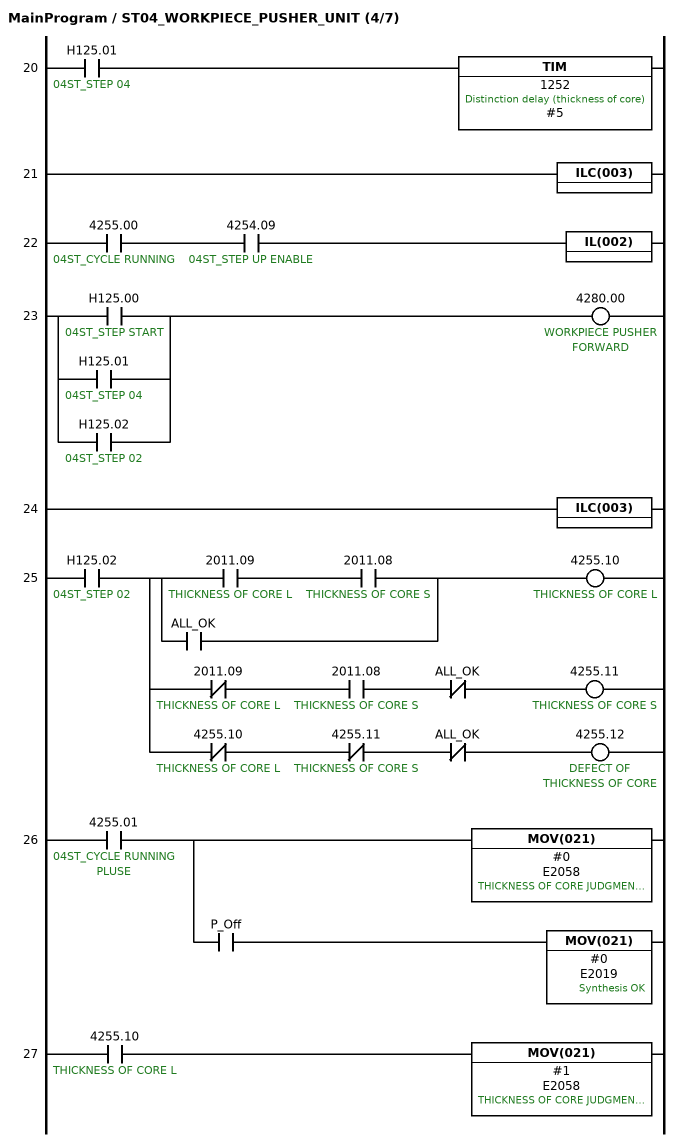
; [picture p336: MainProgram / ST04_WORKPIECE_PUSHER_UNIT, rungs 20-27]
; rung 20
LD H125.01  ; 04ST_STEP 04
TIM 1252 #5  ; Distinction delay (thickness of core)
; rung 21
ILC(003)
; rung 22
LD 4255.00  ; 04ST_CYCLE RUNNING
AND 4254.09  ; 04ST_STEP UP ENABLE
IL(002)
; rung 23
LD H125.00  ; 04ST_STEP START
OR H125.01  ; 04ST_STEP 04
OR H125.02  ; 04ST_STEP 02
OUT 4280.00  ; WORKPIECE PUSHER FORWARD
; rung 24
ILC(003)
; rung 25
LD H125.02  ; 04ST_STEP 02
OUT TR0
LD 2011.09  ; THICKNESS OF CORE L
AND 2011.08  ; THICKNESS OF CORE S
OR ALL_OK
ANDLD
OUT 4255.10  ; THICKNESS OF CORE L
LD TR0
ANDNOT 2011.09  ; THICKNESS OF CORE L
AND 2011.08  ; THICKNESS OF CORE S
ANDNOT ALL_OK
OUT 4255.11  ; THICKNESS OF CORE S
LD TR0
ANDNOT 4255.10  ; THICKNESS OF CORE L
ANDNOT 4255.11  ; THICKNESS OF CORE S
ANDNOT ALL_OK
OUT 4255.12  ; DEFECT OF THICKNESS OF CORE
; rung 26
LD 4255.01  ; 04ST_CYCLE RUNNING PLUSE
MOV(021) #0 E2058  ; THICKNESS OF CORE JUDGMENT RESULT (1:L , 2: S)
AND P_Off
MOV(021) #0 E2019  ; Synthesis OK
; rung 27
LD 4255.10  ; THICKNESS OF CORE L
MOV(021) #1 E2058  ; THICKNESS OF CORE JUDGMENT RESULT (1:L , 2: S)

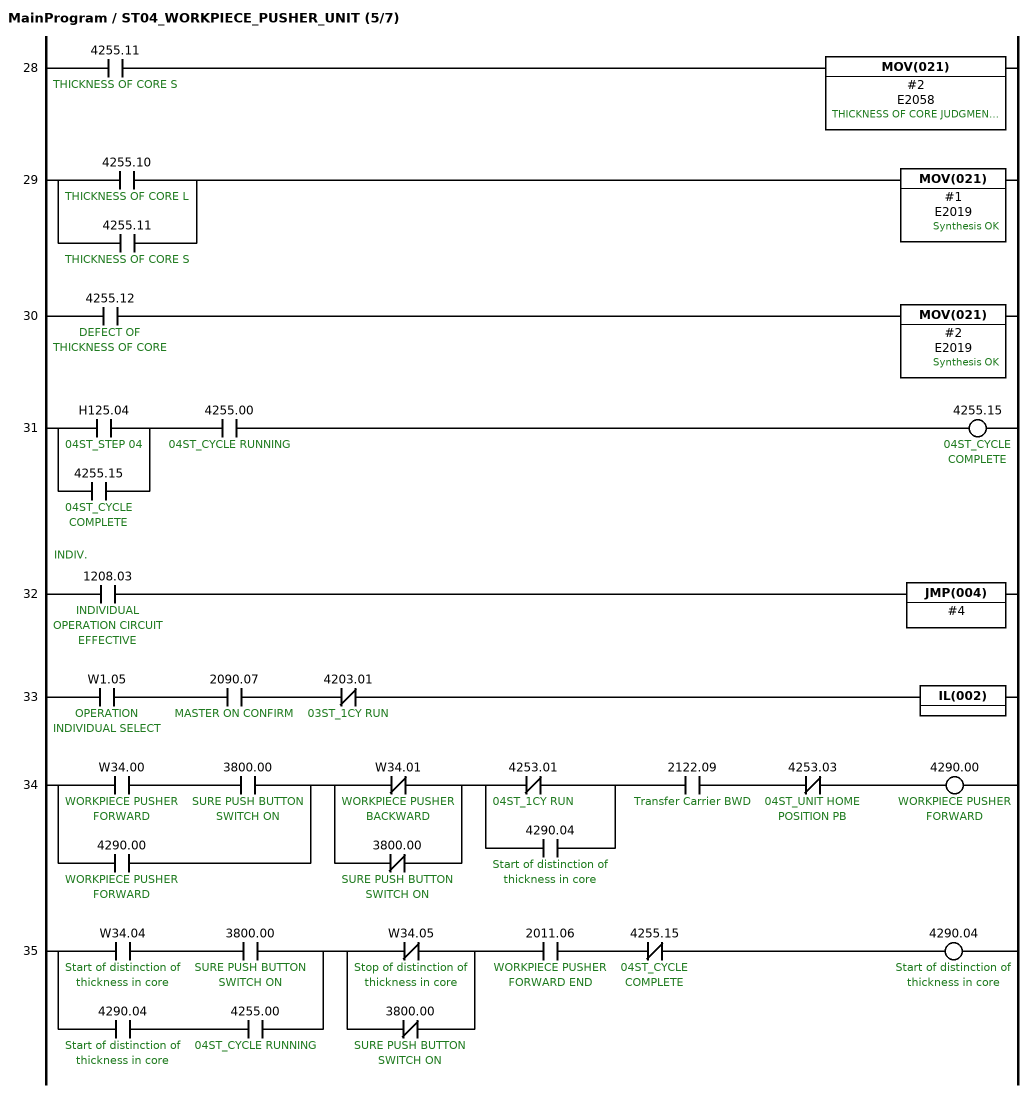
; rung 28
LD 4255.11  ; THICKNESS OF CORE S
MOV(021) #2 E2058  ; THICKNESS OF CORE JUDGMENT RESULT (1:L , 2: S)
; rung 29
LD 4255.10  ; THICKNESS OF CORE L
OR 4255.11  ; THICKNESS OF CORE S
MOV(021) #1 E2019  ; Synthesis OK
; rung 30
LD 4255.12  ; DEFECT OF THICKNESS OF CORE
MOV(021) #2 E2019  ; Synthesis OK
; rung 31
LD H125.04  ; 04ST_STEP 04
OR 4255.15  ; 04ST_CYCLE COMPLETE
AND 4255.00  ; 04ST_CYCLE RUNNING
OUT 4255.15  ; 04ST_CYCLE COMPLETE
; rung 32: INDIV.
LD 1208.03  ; INDIVIDUAL OPERATION CIRCUIT EFFECTIVE
JMP(004) #4
; rung 33
LD W1.05  ; OPERATION INDIVIDUAL SELECT
AND 2090.07  ; MASTER ON CONFIRM
ANDNOT 4203.01  ; 03ST_1CY RUN
IL(002)
; rung 34
LD W34.00  ; WORKPIECE PUSHER FORWARD
AND 3800.00  ; SURE PUSH BUTTON SWITCH ON
OR 4290.00  ; WORKPIECE PUSHER FORWARD
LDNOT W34.01  ; WORKPIECE PUSHER BACKWARD
ORNOT 3800.00  ; SURE PUSH BUTTON SWITCH ON
ANDLD
LDNOT 4253.01  ; 04ST_1CY RUN
OR 4290.04  ; Start of distinction of thickness in core
ANDLD
AND 2122.09  ; Transfer Carrier BWD
ANDNOT 4253.03  ; 04ST_UNIT HOME POSITION PB
OUT 4290.00  ; WORKPIECE PUSHER FORWARD
; rung 35
LD W34.04  ; Start of distinction of thickness in core
AND 3800.00  ; SURE PUSH BUTTON SWITCH ON
LD 4290.04  ; Start of distinction of thickness in core
AND 4255.00  ; 04ST_CYCLE RUNNING
ORLD
LDNOT W34.05  ; Stop of distinction of thickness in core
ORNOT 3800.00  ; SURE PUSH BUTTON SWITCH ON
ANDLD
AND 2011.06  ; WORKPIECE PUSHER FORWARD END
ANDNOT 4255.15  ; 04ST_CYCLE COMPLETE
OUT 4290.04  ; Start of distinction of thickness in core

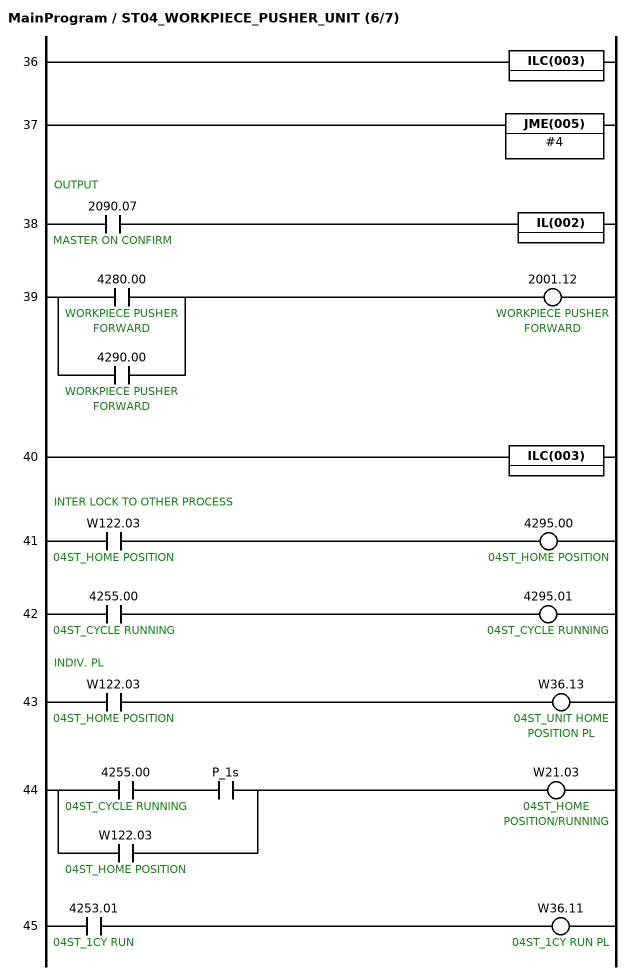
; rung 36
ILC(003)
; rung 37
JME(005) #4
; rung 38: OUTPUT
LD 2090.07  ; MASTER ON CONFIRM
IL(002)
; rung 39
LD 4280.00  ; WORKPIECE PUSHER FORWARD
OR 4290.00  ; WORKPIECE PUSHER FORWARD
OUT 2001.12  ; WORKPIECE PUSHER FORWARD
; rung 40
ILC(003)
; rung 41: INTER LOCK TO OTHER PROCESS
LD W122.03  ; 04ST_HOME POSITION
OUT 4295.00  ; 04ST_HOME POSITION
; rung 42
LD 4255.00  ; 04ST_CYCLE RUNNING
OUT 4295.01  ; 04ST_CYCLE RUNNING
; rung 43: INDIV. PL
LD W122.03  ; 04ST_HOME POSITION
OUT W36.13  ; 04ST_UNIT HOME POSITION PL
; rung 44
LD 4255.00  ; 04ST_CYCLE RUNNING
AND P_1s
OR W122.03  ; 04ST_HOME POSITION
OUT W21.03  ; 04ST_HOME POSITION/RUNNING
; rung 45
LD 4253.01  ; 04ST_1CY RUN
OUT W36.11  ; 04ST_1CY RUN PL

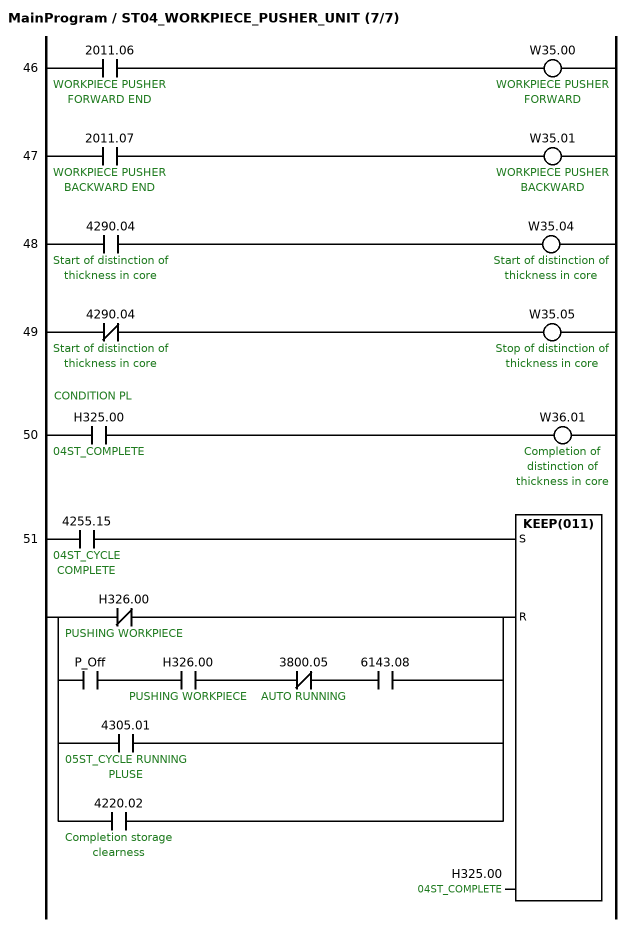
; rung 46
LD 2011.06  ; WORKPIECE PUSHER FORWARD END
OUT W35.00  ; WORKPIECE PUSHER FORWARD
; rung 47
LD 2011.07  ; WORKPIECE PUSHER BACKWARD END
OUT W35.01  ; WORKPIECE PUSHER BACKWARD
; rung 48
LD 4290.04  ; Start of distinction of thickness in core
OUT W35.04  ; Start of distinction of thickness in core
; rung 49
LDNOT 4290.04  ; Start of distinction of thickness in core
OUT W35.05  ; Stop of distinction of thickness in core
; rung 50: CONDITION PL
LD H325.00  ; 04ST_COMPLETE
OUT W36.01  ; Completion of distinction of thickness in core
; rung 51
LD 4255.15  ; 04ST_CYCLE COMPLETE
LDNOT H326.00  ; PUSHING WORKPIECE
LD P_Off
AND H326.00  ; PUSHING WORKPIECE
ANDNOT 3800.05  ; AUTO RUNNING
AND 6143.08
ORLD
OR 4305.01  ; 05ST_CYCLE RUNNING PLUSE
OR 4220.02  ; Completion storage clearness
KEEP(011) H325.00  ; 04ST_COMPLETE

### Section ST05_INSULATION_TEST_UNIT

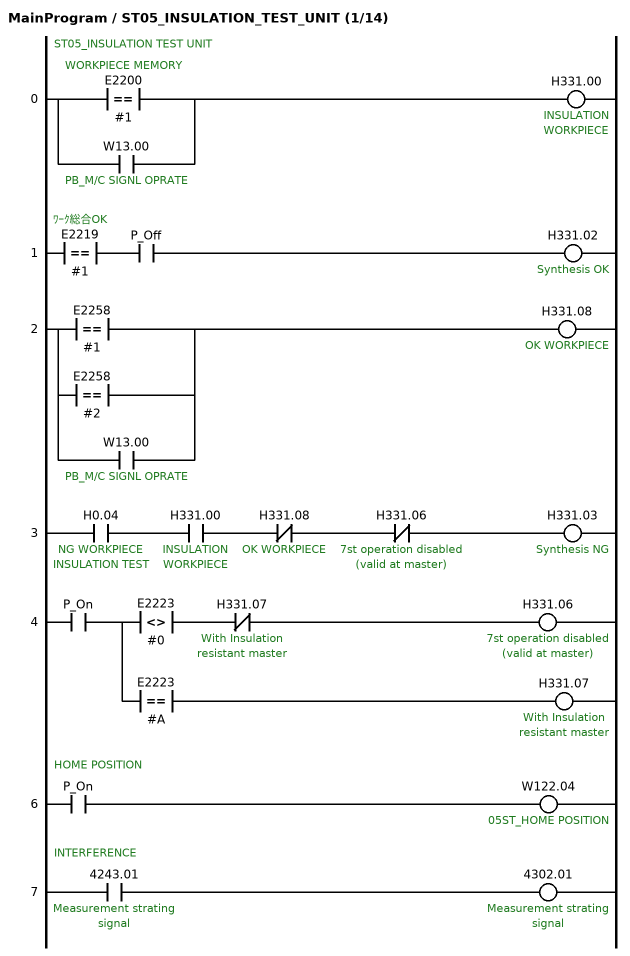
; rung 0: ST05_INSULATION TEST UNIT
LD=(300) E2200 #1  ; WORKPIECE MEMORY
OR W13.00  ; PB_M/C SIGNL OPRATE
OUT H331.00  ; INSULATION WORKPIECE
; rung 1
LD=(300) E2219 #1  ; ﾜｰｸ総合OK
AND P_Off
OUT H331.02  ; Synthesis OK
; rung 2
LD=(300) E2258 #1
OR=(300) E2258 #2
OR W13.00  ; PB_M/C SIGNL OPRATE
OUT H331.08  ; OK WORKPIECE
; rung 3
LD H0.04  ; NG WORKPIECE INSULATION TEST
AND H331.00  ; INSULATION WORKPIECE
ANDNOT H331.08  ; OK WORKPIECE
ANDNOT H331.06  ; 7st operation disabled (valid at master)
OUT H331.03  ; Synthesis NG
; rung 4
LD P_On
OUT TR0
AND<>(305) E2223 #0
ANDNOT H331.07  ; With Insulation resistant master
OUT H331.06  ; 7st operation disabled (valid at master)
LD TR0
AND=(300) E2223 #A
OUT H331.07  ; With Insulation resistant master
; rung 5: TIMER
; rung 6: HOME POSITION
LD P_On
OUT W122.04  ; 05ST_HOME POSITION
; rung 7: INTERFERENCE
LD 4243.01  ; Measurement strating signal
OUT 4302.01  ; Measurement strating signal

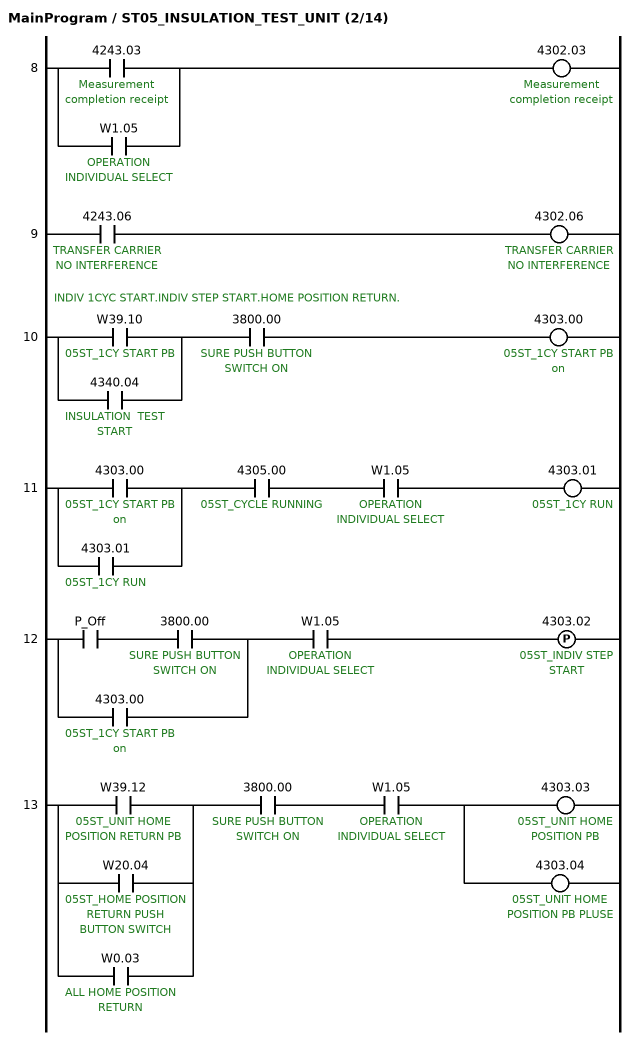
; rung 8
LD 4243.03  ; Measurement completion receipt
OR W1.05  ; OPERATION INDIVIDUAL SELECT
OUT 4302.03  ; Measurement completion receipt
; rung 9
LD 4243.06  ; TRANSFER CARRIER NO INTERFERENCE
OUT 4302.06  ; TRANSFER CARRIER NO INTERFERENCE
; rung 10: INDIV 1CYC START.INDIV STEP START.HOME POSITION RETURN.
LD W39.10  ; 05ST_1CY START PB
OR 4340.04  ; INSULATION  TEST START
AND 3800.00  ; SURE PUSH BUTTON SWITCH ON
OUT 4303.00  ; 05ST_1CY START PB on
; rung 11
LD 4303.00  ; 05ST_1CY START PB on
OR 4303.01  ; 05ST_1CY RUN
AND 4305.00  ; 05ST_CYCLE RUNNING
AND W1.05  ; OPERATION INDIVIDUAL SELECT
OUT 4303.01  ; 05ST_1CY RUN
; rung 12
LD P_Off
AND 3800.00  ; SURE PUSH BUTTON SWITCH ON
OR 4303.00  ; 05ST_1CY START PB on
AND W1.05  ; OPERATION INDIVIDUAL SELECT
DIFU(013) 4303.02  ; 05ST_INDIV STEP START
; rung 13
LD W39.12  ; 05ST_UNIT HOME POSITION RETURN PB
OR W20.04  ; 05ST_HOME POSITION RETURN PUSH BUTTON SWITCH
OR W0.03  ; ALL HOME POSITION RETURN
AND 3800.00  ; SURE PUSH BUTTON SWITCH ON
AND W1.05  ; OPERATION INDIVIDUAL SELECT
OUT 4303.03  ; 05ST_UNIT HOME POSITION PB
OUT 4303.04  ; 05ST_UNIT HOME POSITION PB PLUSE

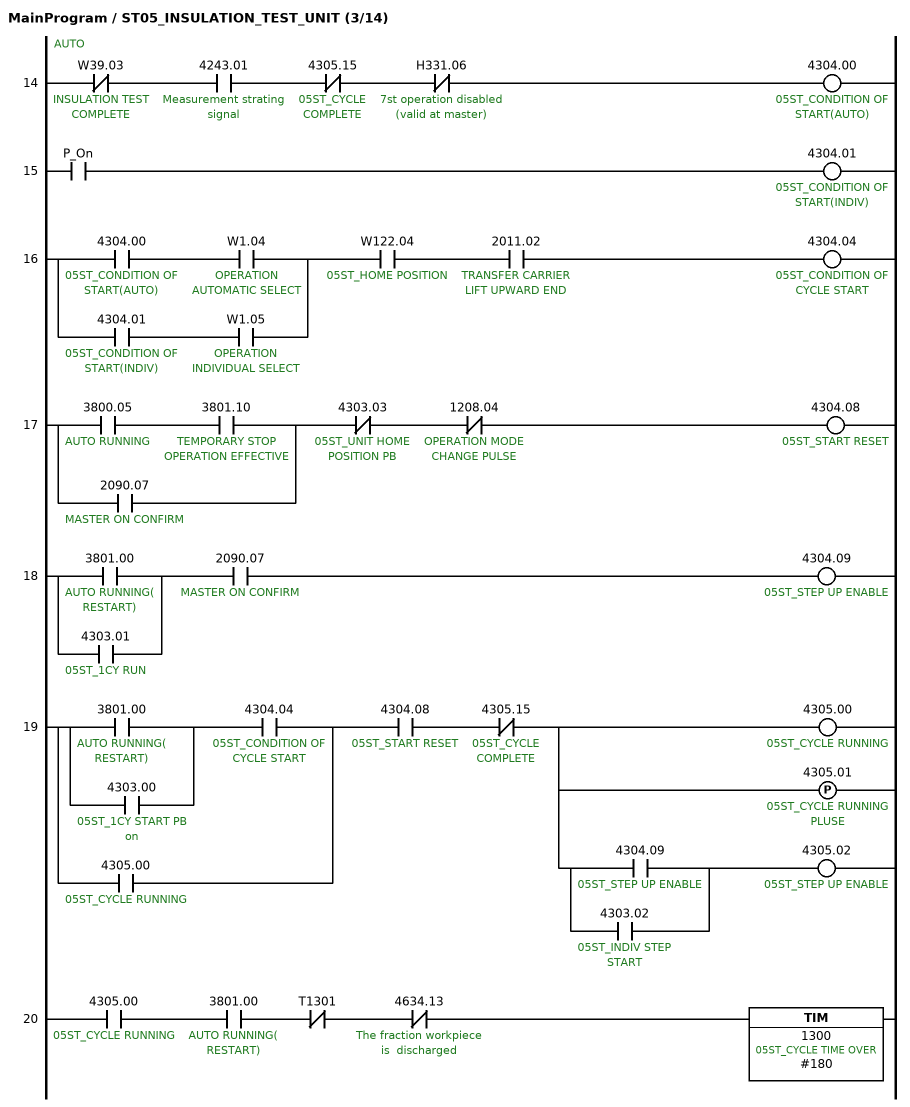
; rung 14: AUTO
LDNOT W39.03  ; INSULATION TEST COMPLETE
AND 4243.01  ; Measurement strating signal
ANDNOT 4305.15  ; 05ST_CYCLE COMPLETE
ANDNOT H331.06  ; 7st operation disabled (valid at master)
OUT 4304.00  ; 05ST_CONDITION OF START(AUTO)
; rung 15
LD P_On
OUT 4304.01  ; 05ST_CONDITION OF START(INDIV)
; rung 16
LD 4304.00  ; 05ST_CONDITION OF START(AUTO)
AND W1.04  ; OPERATION AUTOMATIC SELECT
LD 4304.01  ; 05ST_CONDITION OF START(INDIV)
AND W1.05  ; OPERATION INDIVIDUAL SELECT
ORLD
AND W122.04  ; 05ST_HOME POSITION
AND 2011.02  ; TRANSFER CARRIER LIFT UPWARD END
OUT 4304.04  ; 05ST_CONDITION OF CYCLE START
; rung 17
LD 3800.05  ; AUTO RUNNING
AND 3801.10  ; TEMPORARY STOP OPERATION EFFECTIVE
OR 2090.07  ; MASTER ON CONFIRM
ANDNOT 4303.03  ; 05ST_UNIT HOME POSITION PB
ANDNOT 1208.04  ; OPERATION MODE CHANGE PULSE
OUT 4304.08  ; 05ST_START RESET
; rung 18
LD 3801.00  ; AUTO RUNNING(RESTART)
OR 4303.01  ; 05ST_1CY RUN
AND 2090.07  ; MASTER ON CONFIRM
OUT 4304.09  ; 05ST_STEP UP ENABLE
; rung 19
LD 3801.00  ; AUTO RUNNING(RESTART)
OR 4303.00  ; 05ST_1CY START PB on
AND 4304.04  ; 05ST_CONDITION OF CYCLE START
OR 4305.00  ; 05ST_CYCLE RUNNING
AND 4304.08  ; 05ST_START RESET
ANDNOT 4305.15  ; 05ST_CYCLE COMPLETE
OUT 4305.00  ; 05ST_CYCLE RUNNING
DIFU(013) 4305.01  ; 05ST_CYCLE RUNNING PLUSE
LD 4304.09  ; 05ST_STEP UP ENABLE
OR 4303.02  ; 05ST_INDIV STEP START
ANDLD
OUT 4305.02  ; 05ST_STEP UP ENABLE
; rung 20
LD 4305.00  ; 05ST_CYCLE RUNNING
AND 3801.00  ; AUTO RUNNING(RESTART)
ANDNOT T1301
ANDNOT 4634.13  ; The fraction workpiece is  discharged
TIM 1300 #180  ; 05ST_CYCLE TIME OVER

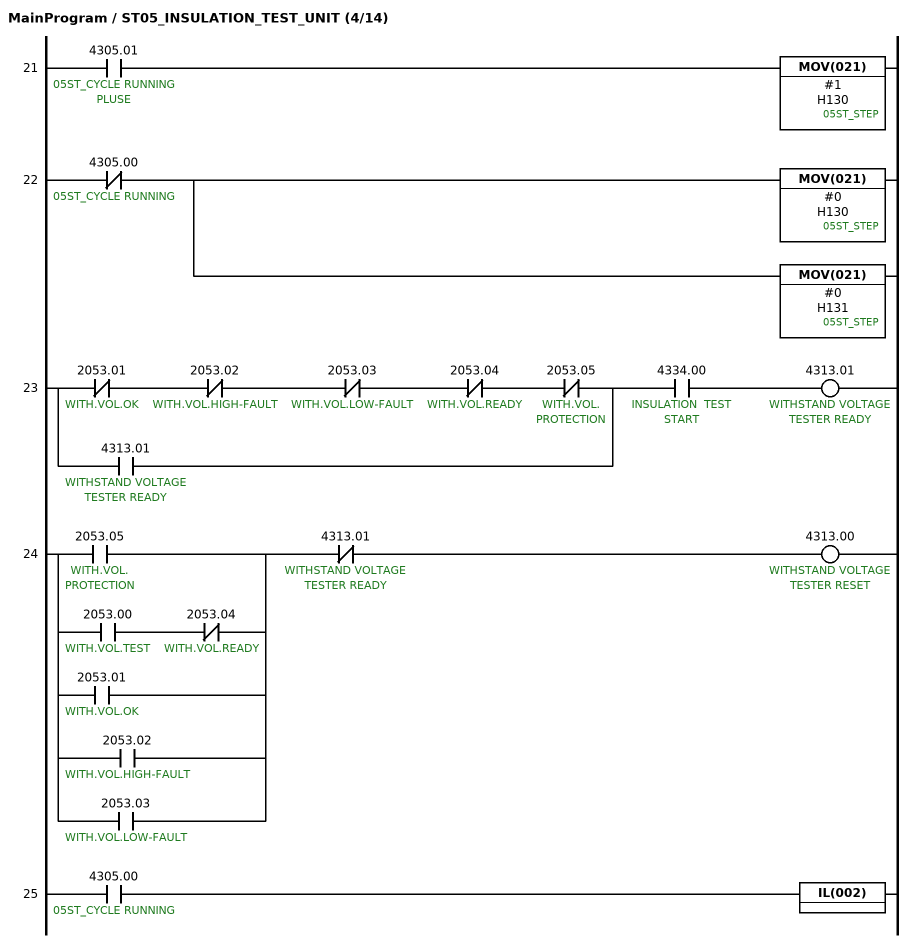
; rung 21
LD 4305.01  ; 05ST_CYCLE RUNNING PLUSE
MOV(021) #1 H130  ; 05ST_STEP
; rung 22
LDNOT 4305.00  ; 05ST_CYCLE RUNNING
MOV(021) #0 H130  ; 05ST_STEP
MOV(021) #0 H131  ; 05ST_STEP
; rung 23
LDNOT 2053.01  ; WITH.VOL.OK
ANDNOT 2053.02  ; WITH.VOL.HIGH-FAULT
ANDNOT 2053.03  ; WITH.VOL.LOW-FAULT
ANDNOT 2053.04  ; WITH.VOL.READY
ANDNOT 2053.05  ; WITH.VOL.PROTECTION
OR 4313.01  ; WITHSTAND VOLTAGE TESTER READY
AND 4334.00  ; INSULATION  TEST START
OUT 4313.01  ; WITHSTAND VOLTAGE TESTER READY
; rung 24
LD 2053.05  ; WITH.VOL.PROTECTION
LD 2053.00  ; WITH.VOL.TEST
ANDNOT 2053.04  ; WITH.VOL.READY
ORLD
OR 2053.01  ; WITH.VOL.OK
OR 2053.02  ; WITH.VOL.HIGH-FAULT
OR 2053.03  ; WITH.VOL.LOW-FAULT
ANDNOT 4313.01  ; WITHSTAND VOLTAGE TESTER READY
OUT 4313.00  ; WITHSTAND VOLTAGE TESTER RESET
; rung 25
LD 4305.00  ; 05ST_CYCLE RUNNING
IL(002)

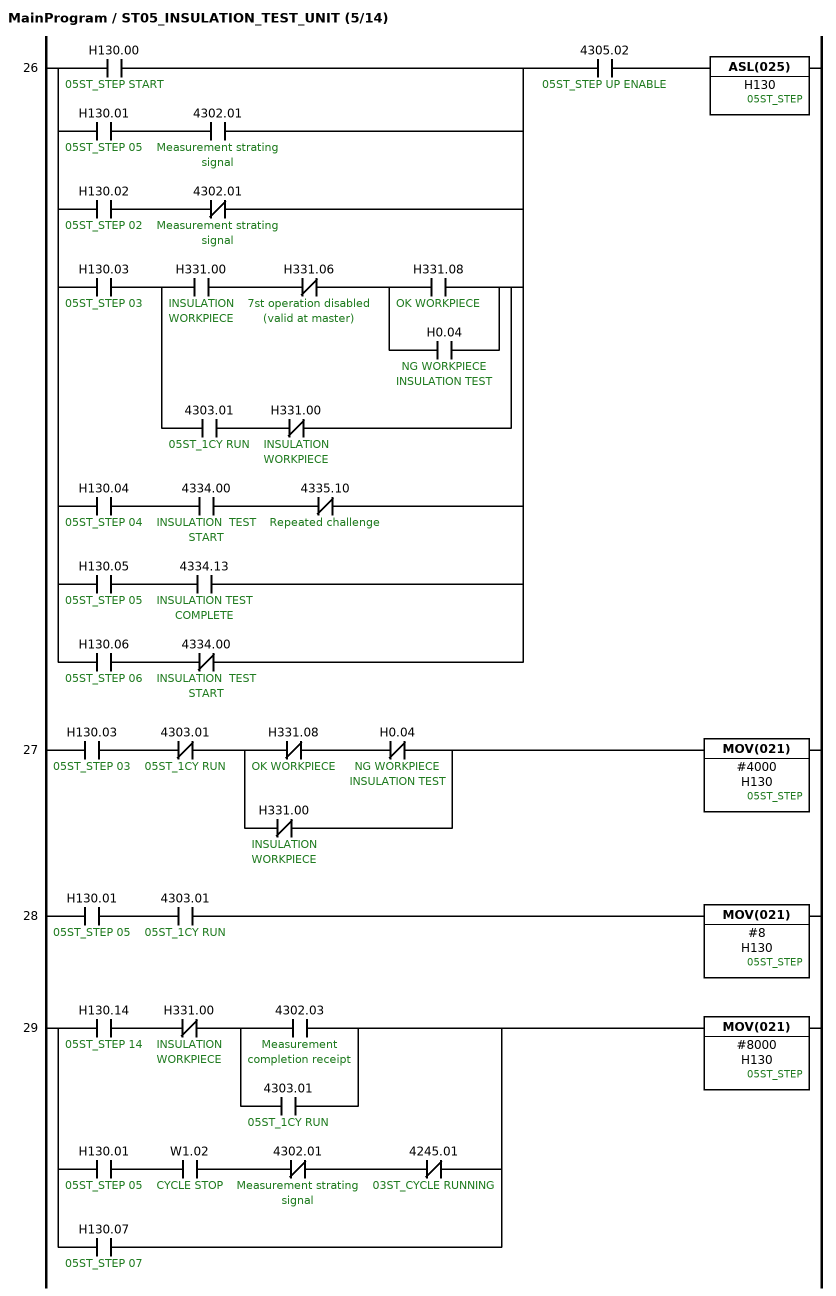
; rung 26
LD H130.00  ; 05ST_STEP START
LD H130.01  ; 05ST_STEP 05
AND 4302.01  ; Measurement strating signal
ORLD
LD H130.02  ; 05ST_STEP 02
ANDNOT 4302.01  ; Measurement strating signal
ORLD
LD H130.03  ; 05ST_STEP 03
LD H331.00  ; INSULATION WORKPIECE
ANDNOT H331.06  ; 7st operation disabled (valid at master)
LD H331.08  ; OK WORKPIECE
OR H0.04  ; NG WORKPIECE INSULATION TEST
ANDLD
LD 4303.01  ; 05ST_1CY RUN
ANDNOT H331.00  ; INSULATION WORKPIECE
ORLD
ANDLD
ORLD
LD H130.04  ; 05ST_STEP 04
AND 4334.00  ; INSULATION  TEST START
ANDNOT 4335.10  ; Repeated challenge
ORLD
LD H130.05  ; 05ST_STEP 05
AND 4334.13  ; INSULATION TEST COMPLETE
ORLD
LD H130.06  ; 05ST_STEP 06
ANDNOT 4334.00  ; INSULATION  TEST START
ORLD
AND 4305.02  ; 05ST_STEP UP ENABLE
ASL(025) H130  ; 05ST_STEP
; rung 27
LD H130.03  ; 05ST_STEP 03
ANDNOT 4303.01  ; 05ST_1CY RUN
LDNOT H331.08  ; OK WORKPIECE
ANDNOT H0.04  ; NG WORKPIECE INSULATION TEST
ORNOT H331.00  ; INSULATION WORKPIECE
ANDLD
MOV(021) #4000 H130  ; 05ST_STEP
; rung 28
LD H130.01  ; 05ST_STEP 05
AND 4303.01  ; 05ST_1CY RUN
MOV(021) #8 H130  ; 05ST_STEP
; rung 29
LD H130.14  ; 05ST_STEP 14
ANDNOT H331.00  ; INSULATION WORKPIECE
LD 4302.03  ; Measurement completion receipt
OR 4303.01  ; 05ST_1CY RUN
ANDLD
LD H130.01  ; 05ST_STEP 05
AND W1.02  ; CYCLE STOP
ANDNOT 4302.01  ; Measurement strating signal
ANDNOT 4245.01  ; 03ST_CYCLE RUNNING
ORLD
OR H130.07  ; 05ST_STEP 07
MOV(021) #8000 H130  ; 05ST_STEP

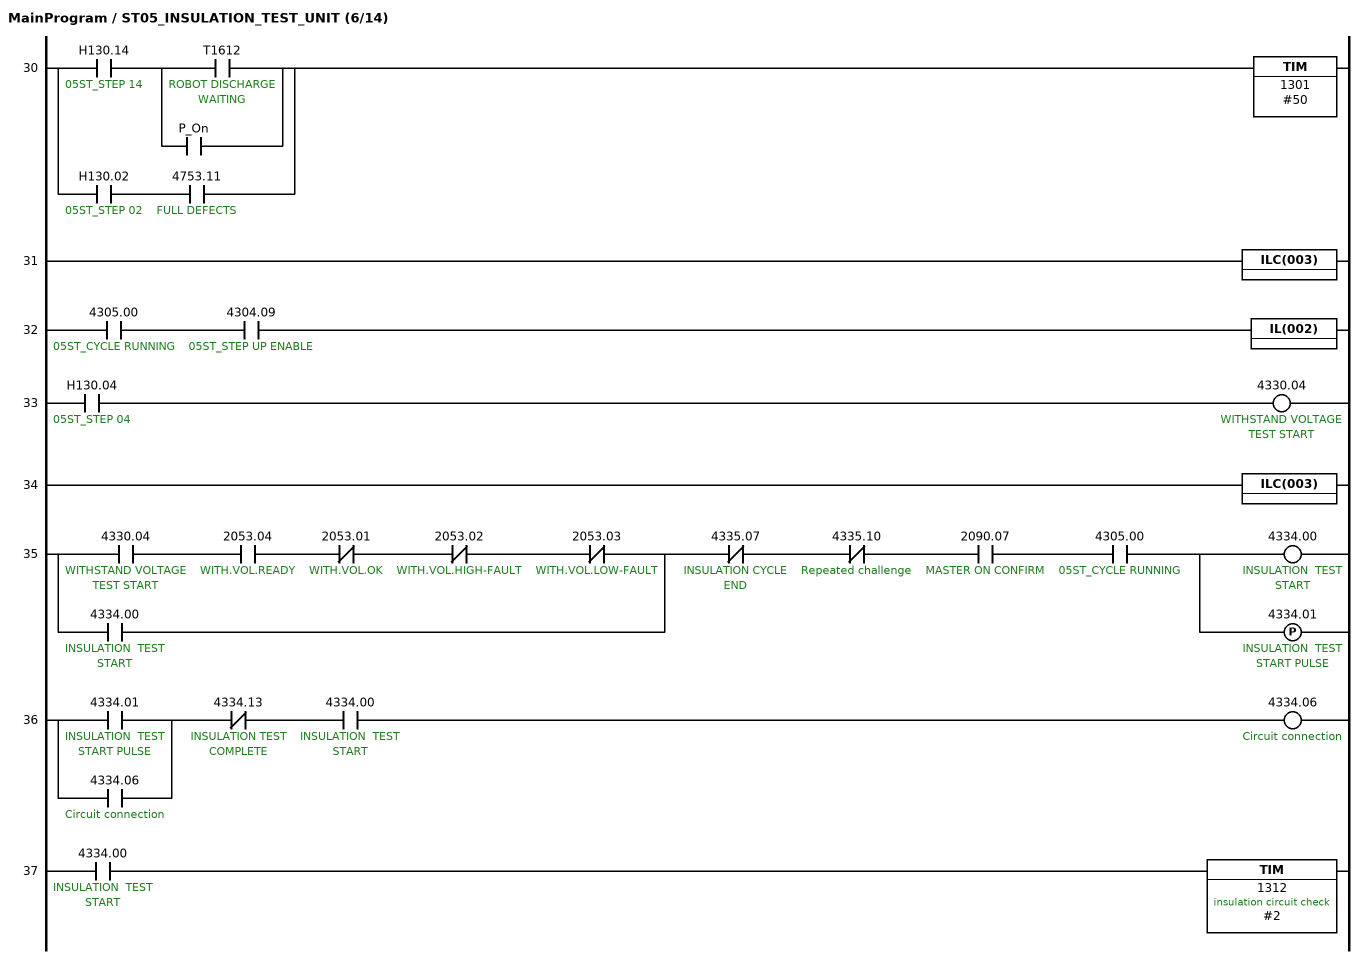
; rung 30
LD H130.14  ; 05ST_STEP 14
LD T1612  ; ROBOT DISCHARGE WAITING
OR P_On
ANDLD
LD H130.02  ; 05ST_STEP 02
AND 4753.11  ; FULL DEFECTS
ORLD
TIM 1301 #50
; rung 31
ILC(003)
; rung 32
LD 4305.00  ; 05ST_CYCLE RUNNING
AND 4304.09  ; 05ST_STEP UP ENABLE
IL(002)
; rung 33
LD H130.04  ; 05ST_STEP 04
OUT 4330.04  ; WITHSTAND VOLTAGE TEST START
; rung 34
ILC(003)
; rung 35
LD 4330.04  ; WITHSTAND VOLTAGE TEST START
AND 2053.04  ; WITH.VOL.READY
ANDNOT 2053.01  ; WITH.VOL.OK
ANDNOT 2053.02  ; WITH.VOL.HIGH-FAULT
ANDNOT 2053.03  ; WITH.VOL.LOW-FAULT
OR 4334.00  ; INSULATION  TEST START
ANDNOT 4335.07  ; INSULATION CYCLE END
ANDNOT 4335.10  ; Repeated challenge
AND 2090.07  ; MASTER ON CONFIRM
AND 4305.00  ; 05ST_CYCLE RUNNING
OUT 4334.00  ; INSULATION  TEST START
DIFU(013) 4334.01  ; INSULATION  TEST START PULSE
; rung 36
LD 4334.01  ; INSULATION  TEST START PULSE
OR 4334.06  ; Circuit connection
ANDNOT 4334.13  ; INSULATION TEST COMPLETE
AND 4334.00  ; INSULATION  TEST START
OUT 4334.06  ; Circuit connection
; rung 37
LD 4334.00  ; INSULATION  TEST START
TIM 1312 #2  ; insulation circuit check

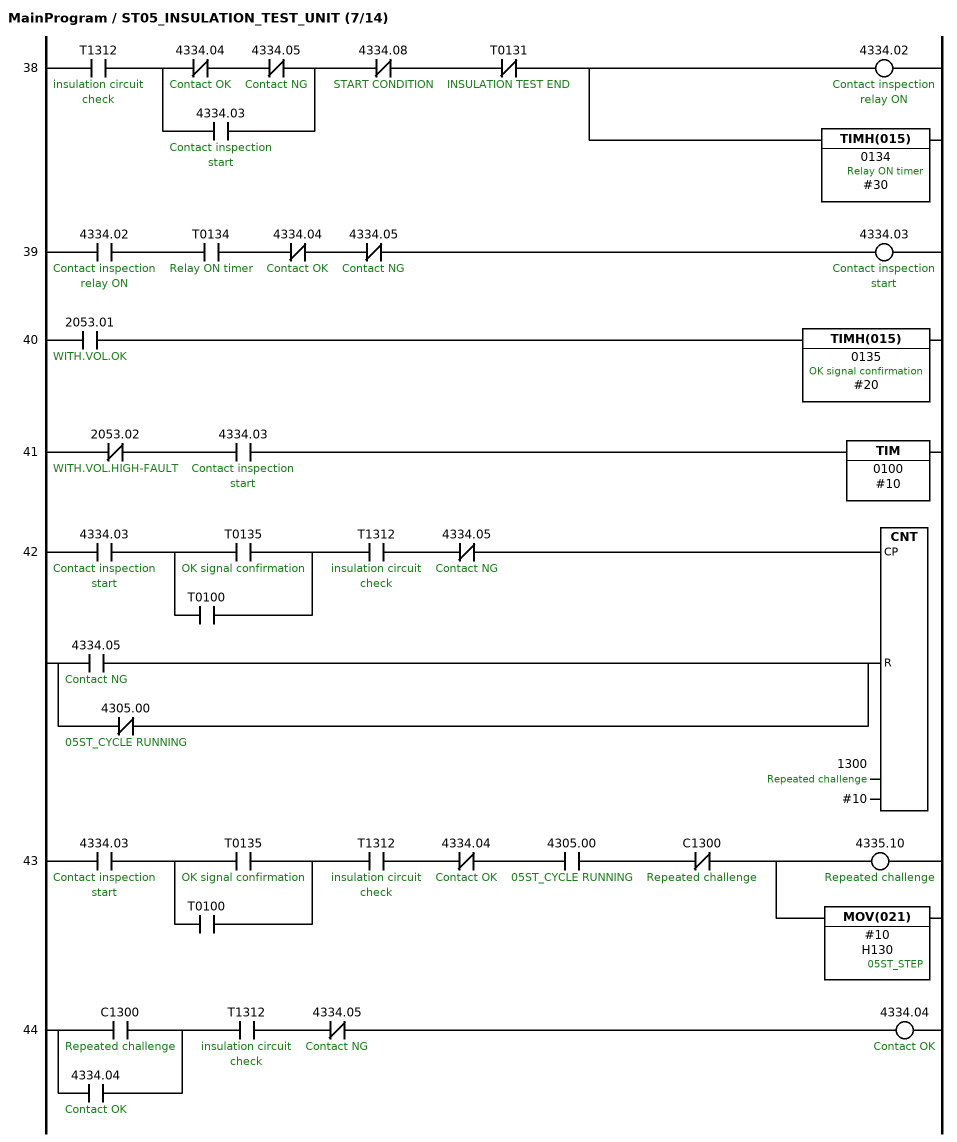
; rung 38
LD T1312  ; insulation circuit check
LDNOT 4334.04  ; Contact OK
ANDNOT 4334.05  ; Contact NG
OR 4334.03  ; Contact inspection start
ANDLD
ANDNOT 4334.08  ; START CONDITION
ANDNOT T0131  ; INSULATION TEST END
OUT 4334.02  ; Contact inspection relay ON
TIMH(015) 0134 #30  ; Relay ON timer
; rung 39
LD 4334.02  ; Contact inspection relay ON
AND T0134  ; Relay ON timer
ANDNOT 4334.04  ; Contact OK
ANDNOT 4334.05  ; Contact NG
OUT 4334.03  ; Contact inspection start
; rung 40
LD 2053.01  ; WITH.VOL.OK
TIMH(015) 0135 #20  ; OK signal confirmation
; rung 41
LDNOT 2053.02  ; WITH.VOL.HIGH-FAULT
AND 4334.03  ; Contact inspection start
TIM 0100 #10
; rung 42
LD 4334.03  ; Contact inspection start
LD T0135  ; OK signal confirmation
OR T0100
ANDLD
AND T1312  ; insulation circuit check
ANDNOT 4334.05  ; Contact NG
LD 4334.05  ; Contact NG
ORNOT 4305.00  ; 05ST_CYCLE RUNNING
CNT 1300 #10  ; Repeated challenge
; rung 43
LD 4334.03  ; Contact inspection start
LD T0135  ; OK signal confirmation
OR T0100
ANDLD
AND T1312  ; insulation circuit check
ANDNOT 4334.04  ; Contact OK
AND 4305.00  ; 05ST_CYCLE RUNNING
ANDNOT C1300  ; Repeated challenge
OUT 4335.10  ; Repeated challenge
MOV(021) #10 H130  ; 05ST_STEP
; rung 44
LD C1300  ; Repeated challenge
OR 4334.04  ; Contact OK
AND T1312  ; insulation circuit check
ANDNOT 4334.05  ; Contact NG
OUT 4334.04  ; Contact OK

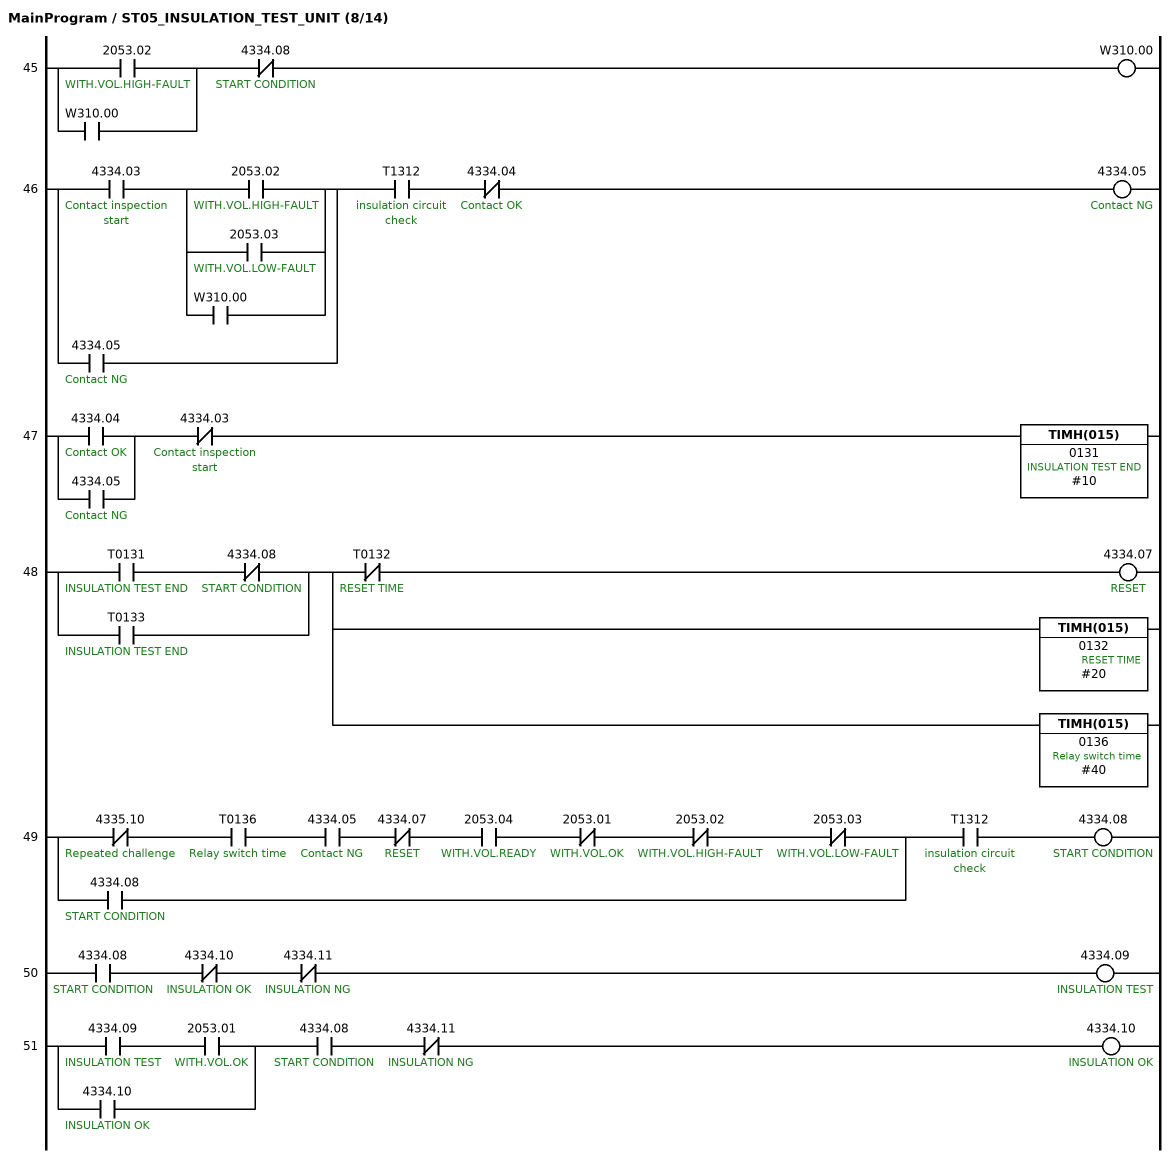
; rung 45
LD 2053.02  ; WITH.VOL.HIGH-FAULT
OR W310.00
ANDNOT 4334.08  ; START CONDITION
OUT W310.00
; rung 46
LD 4334.03  ; Contact inspection start
LD 2053.02  ; WITH.VOL.HIGH-FAULT
OR 2053.03  ; WITH.VOL.LOW-FAULT
OR W310.00
ANDLD
OR 4334.05  ; Contact NG
AND T1312  ; insulation circuit check
ANDNOT 4334.04  ; Contact OK
OUT 4334.05  ; Contact NG
; rung 47
LD 4334.04  ; Contact OK
OR 4334.05  ; Contact NG
ANDNOT 4334.03  ; Contact inspection start
TIMH(015) 0131 #10  ; INSULATION TEST END
; rung 48
LD T0131  ; INSULATION TEST END
ANDNOT 4334.08  ; START CONDITION
OR T0133  ; INSULATION TEST END
OUT TR0
ANDNOT T0132  ; RESET TIME
OUT 4334.07  ; RESET
LD TR0
TIMH(015) 0132 #20  ; RESET TIME
TIMH(015) 0136 #40  ; Relay switch time
; rung 49
LDNOT 4335.10  ; Repeated challenge
AND T0136  ; Relay switch time
AND 4334.05  ; Contact NG
ANDNOT 4334.07  ; RESET
AND 2053.04  ; WITH.VOL.READY
ANDNOT 2053.01  ; WITH.VOL.OK
ANDNOT 2053.02  ; WITH.VOL.HIGH-FAULT
ANDNOT 2053.03  ; WITH.VOL.LOW-FAULT
OR 4334.08  ; START CONDITION
AND T1312  ; insulation circuit check
OUT 4334.08  ; START CONDITION
; rung 50
LD 4334.08  ; START CONDITION
ANDNOT 4334.10  ; INSULATION OK
ANDNOT 4334.11  ; INSULATION NG
OUT 4334.09  ; INSULATION TEST
; rung 51
LD 4334.09  ; INSULATION TEST
AND 2053.01  ; WITH.VOL.OK
OR 4334.10  ; INSULATION OK
AND 4334.08  ; START CONDITION
ANDNOT 4334.11  ; INSULATION NG
OUT 4334.10  ; INSULATION OK

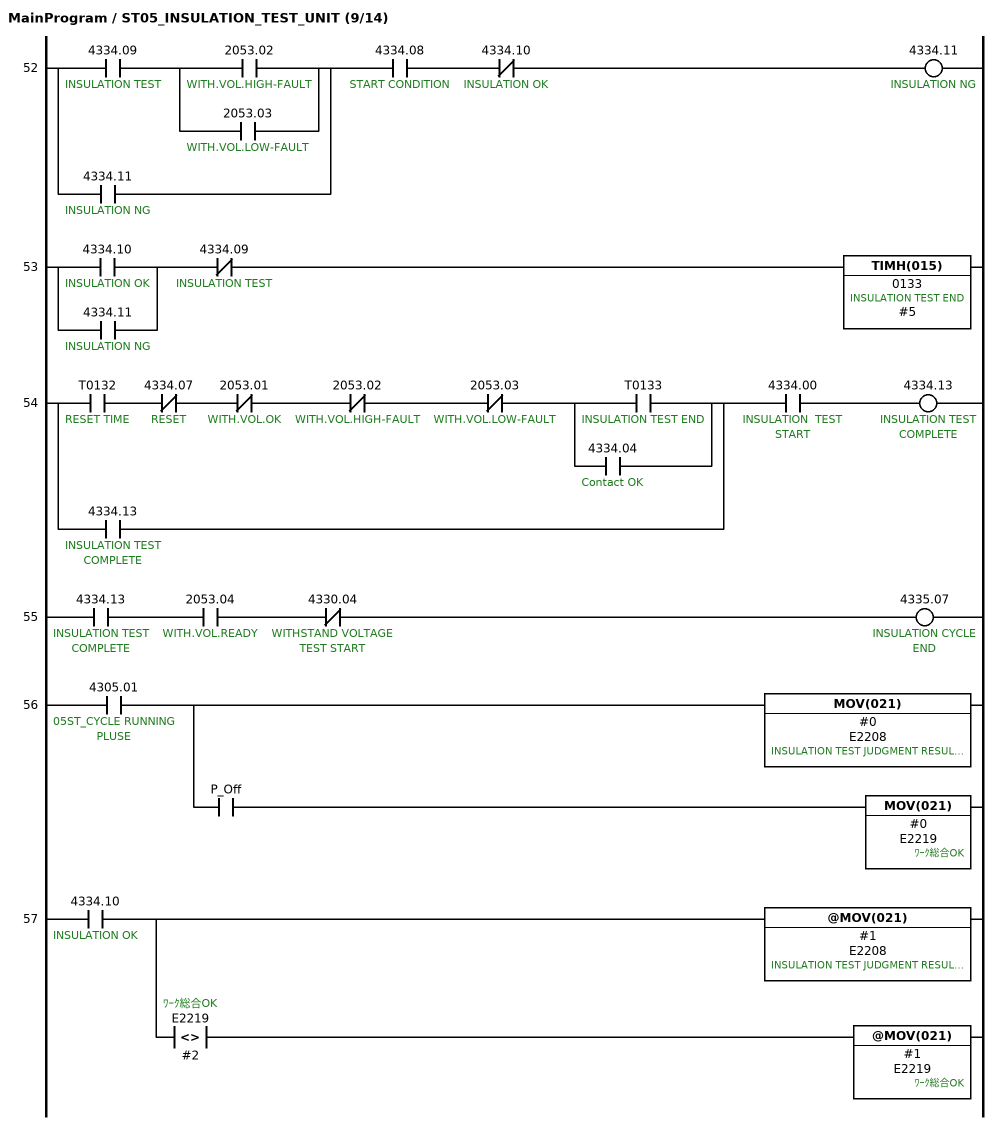
; rung 52
LD 4334.09  ; INSULATION TEST
LD 2053.02  ; WITH.VOL.HIGH-FAULT
OR 2053.03  ; WITH.VOL.LOW-FAULT
ANDLD
OR 4334.11  ; INSULATION NG
AND 4334.08  ; START CONDITION
ANDNOT 4334.10  ; INSULATION OK
OUT 4334.11  ; INSULATION NG
; rung 53
LD 4334.10  ; INSULATION OK
OR 4334.11  ; INSULATION NG
ANDNOT 4334.09  ; INSULATION TEST
TIMH(015) 0133 #5  ; INSULATION TEST END
; rung 54
LD T0132  ; RESET TIME
ANDNOT 4334.07  ; RESET
ANDNOT 2053.01  ; WITH.VOL.OK
ANDNOT 2053.02  ; WITH.VOL.HIGH-FAULT
ANDNOT 2053.03  ; WITH.VOL.LOW-FAULT
LD T0133  ; INSULATION TEST END
OR 4334.04  ; Contact OK
ANDLD
OR 4334.13  ; INSULATION TEST COMPLETE
AND 4334.00  ; INSULATION  TEST START
OUT 4334.13  ; INSULATION TEST COMPLETE
; rung 55
LD 4334.13  ; INSULATION TEST COMPLETE
AND 2053.04  ; WITH.VOL.READY
ANDNOT 4330.04  ; WITHSTAND VOLTAGE TEST START
OUT 4335.07  ; INSULATION CYCLE END
; rung 56
LD 4305.01  ; 05ST_CYCLE RUNNING PLUSE
MOV(021) #0 E2208  ; INSULATION TEST JUDGMENT RESULT (1:OK,2:NG)
AND P_Off
MOV(021) #0 E2219  ; ﾜｰｸ総合OK
; rung 57
LD 4334.10  ; INSULATION OK
@MOV(021) #1 E2208  ; INSULATION TEST JUDGMENT RESULT (1:OK,2:NG)
AND<>(305) E2219 #2  ; ﾜｰｸ総合OK
@MOV(021) #1 E2219  ; ﾜｰｸ総合OK

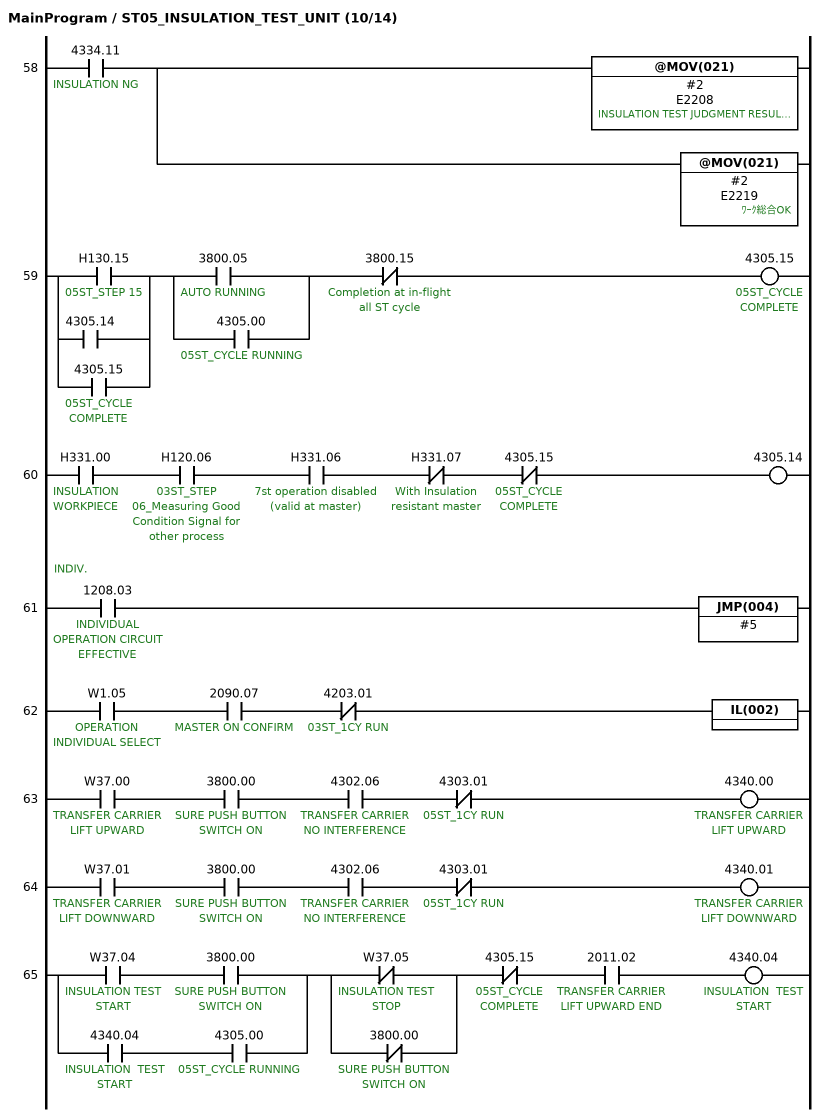
; rung 58
LD 4334.11  ; INSULATION NG
@MOV(021) #2 E2208  ; INSULATION TEST JUDGMENT RESULT (1:OK,2:NG)
@MOV(021) #2 E2219  ; ﾜｰｸ総合OK
; rung 59
LD H130.15  ; 05ST_STEP 15
OR 4305.14
OR 4305.15  ; 05ST_CYCLE COMPLETE
LD 3800.05  ; AUTO RUNNING
OR 4305.00  ; 05ST_CYCLE RUNNING
ANDLD
ANDNOT 3800.15  ; Completion at in-flight all ST cycle
OUT 4305.15  ; 05ST_CYCLE COMPLETE
; rung 60
LD H331.00  ; INSULATION WORKPIECE
AND H120.06  ; 03ST_STEP 06_Measuring Good Condition Signal for other process
AND H331.06  ; 7st operation disabled (valid at master)
ANDNOT H331.07  ; With Insulation resistant master
ANDNOT 4305.15  ; 05ST_CYCLE COMPLETE
OUT 4305.14
; rung 61: INDIV.
LD 1208.03  ; INDIVIDUAL OPERATION CIRCUIT EFFECTIVE
JMP(004) #5
; rung 62
LD W1.05  ; OPERATION INDIVIDUAL SELECT
AND 2090.07  ; MASTER ON CONFIRM
ANDNOT 4203.01  ; 03ST_1CY RUN
IL(002)
; rung 63
LD W37.00  ; TRANSFER CARRIER LIFT UPWARD
AND 3800.00  ; SURE PUSH BUTTON SWITCH ON
AND 4302.06  ; TRANSFER CARRIER NO INTERFERENCE
ANDNOT 4303.01  ; 05ST_1CY RUN
OUT 4340.00  ; TRANSFER CARRIER LIFT UPWARD
; rung 64
LD W37.01  ; TRANSFER CARRIER LIFT DOWNWARD
AND 3800.00  ; SURE PUSH BUTTON SWITCH ON
AND 4302.06  ; TRANSFER CARRIER NO INTERFERENCE
ANDNOT 4303.01  ; 05ST_1CY RUN
OUT 4340.01  ; TRANSFER CARRIER LIFT DOWNWARD
; rung 65
LD W37.04  ; INSULATION TEST START
AND 3800.00  ; SURE PUSH BUTTON SWITCH ON
LD 4340.04  ; INSULATION  TEST START
AND 4305.00  ; 05ST_CYCLE RUNNING
ORLD
LDNOT W37.05  ; INSULATION TEST STOP
ORNOT 3800.00  ; SURE PUSH BUTTON SWITCH ON
ANDLD
ANDNOT 4305.15  ; 05ST_CYCLE COMPLETE
AND 2011.02  ; TRANSFER CARRIER LIFT UPWARD END
OUT 4340.04  ; INSULATION  TEST START

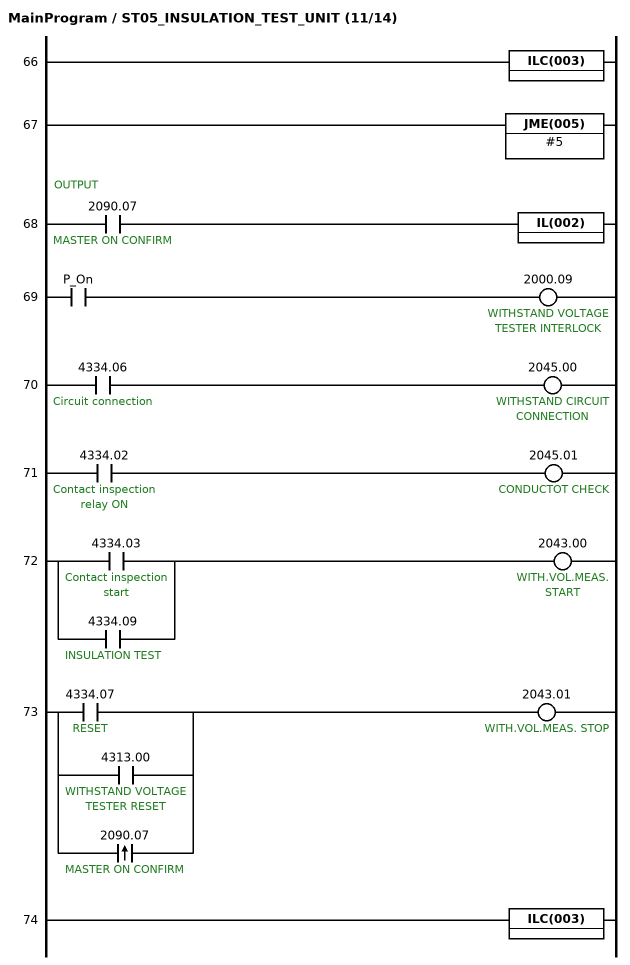
; rung 66
ILC(003)
; rung 67
JME(005) #5
; rung 68: OUTPUT
LD 2090.07  ; MASTER ON CONFIRM
IL(002)
; rung 69
LD P_On
OUT 2000.09  ; WITHSTAND VOLTAGE TESTER INTERLOCK
; rung 70
LD 4334.06  ; Circuit connection
OUT 2045.00  ; WITHSTAND CIRCUIT CONNECTION
; rung 71
LD 4334.02  ; Contact inspection relay ON
OUT 2045.01  ; CONDUCTOT CHECK
; rung 72
LD 4334.03  ; Contact inspection start
OR 4334.09  ; INSULATION TEST
OUT 2043.00  ; WITH.VOL.MEAS. START
; rung 73
LD 4334.07  ; RESET
OR 4313.00  ; WITHSTAND VOLTAGE TESTER RESET
@OR 2090.07  ; MASTER ON CONFIRM
OUT 2043.01  ; WITH.VOL.MEAS. STOP
; rung 74
ILC(003)

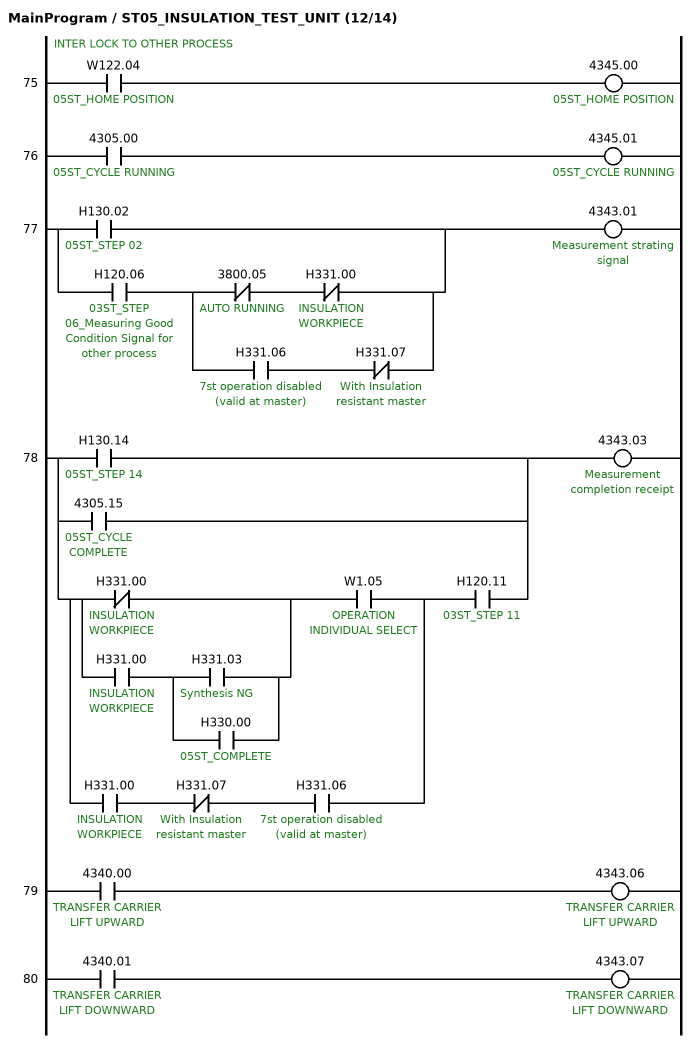
; rung 75: INTER LOCK TO OTHER PROCESS
LD W122.04  ; 05ST_HOME POSITION
OUT 4345.00  ; 05ST_HOME POSITION
; rung 76
LD 4305.00  ; 05ST_CYCLE RUNNING
OUT 4345.01  ; 05ST_CYCLE RUNNING
; rung 77
LD H130.02  ; 05ST_STEP 02
LD H120.06  ; 03ST_STEP 06_Measuring Good Condition Signal for other process
LDNOT 3800.05  ; AUTO RUNNING
ANDNOT H331.00  ; INSULATION WORKPIECE
LD H331.06  ; 7st operation disabled (valid at master)
ANDNOT H331.07  ; With Insulation resistant master
ORLD
ANDLD
ORLD
OUT 4343.01  ; Measurement strating signal
; rung 78
LD H130.14  ; 05ST_STEP 14
OR 4305.15  ; 05ST_CYCLE COMPLETE
LDNOT H331.00  ; INSULATION WORKPIECE
LD H331.00  ; INSULATION WORKPIECE
LD H331.03  ; Synthesis NG
OR H330.00  ; 05ST_COMPLETE
ANDLD
ORLD
AND W1.05  ; OPERATION INDIVIDUAL SELECT
LD H331.00  ; INSULATION WORKPIECE
ANDNOT H331.07  ; With Insulation resistant master
AND H331.06  ; 7st operation disabled (valid at master)
ORLD
AND H120.11  ; 03ST_STEP 11
ORLD
OUT 4343.03  ; Measurement completion receipt
; rung 79
LD 4340.00  ; TRANSFER CARRIER LIFT UPWARD
OUT 4343.06  ; TRANSFER CARRIER LIFT UPWARD
; rung 80
LD 4340.01  ; TRANSFER CARRIER LIFT DOWNWARD
OUT 4343.07  ; TRANSFER CARRIER LIFT DOWNWARD

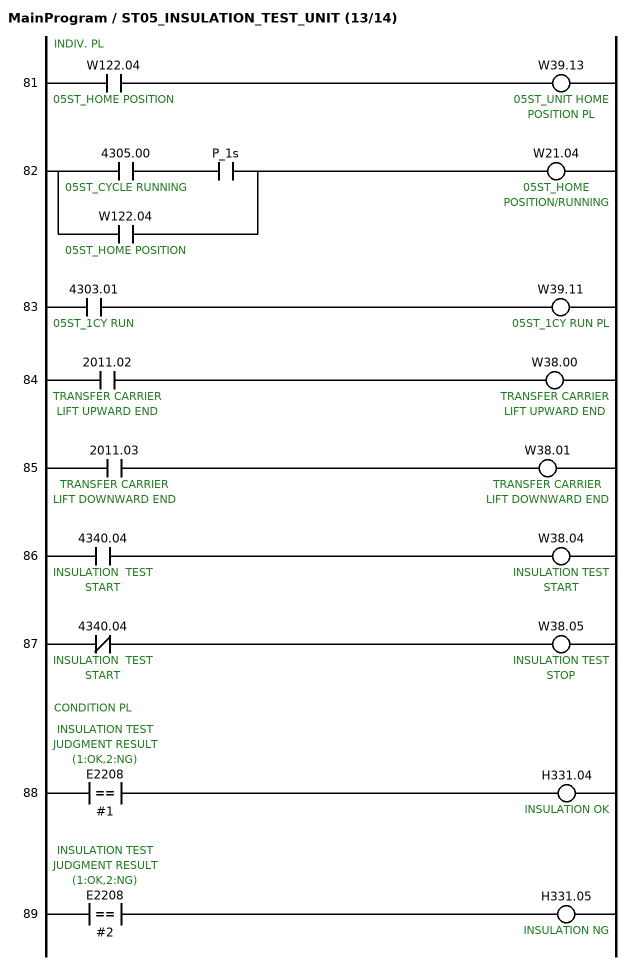
; rung 81: INDIV. PL
LD W122.04  ; 05ST_HOME POSITION
OUT W39.13  ; 05ST_UNIT HOME POSITION PL
; rung 82
LD 4305.00  ; 05ST_CYCLE RUNNING
AND P_1s
OR W122.04  ; 05ST_HOME POSITION
OUT W21.04  ; 05ST_HOME POSITION/RUNNING
; rung 83
LD 4303.01  ; 05ST_1CY RUN
OUT W39.11  ; 05ST_1CY RUN PL
; rung 84
LD 2011.02  ; TRANSFER CARRIER LIFT UPWARD END
OUT W38.00  ; TRANSFER CARRIER LIFT UPWARD END
; rung 85
LD 2011.03  ; TRANSFER CARRIER LIFT DOWNWARD END
OUT W38.01  ; TRANSFER CARRIER LIFT DOWNWARD END
; rung 86
LD 4340.04  ; INSULATION  TEST START
OUT W38.04  ; INSULATION TEST START
; rung 87
LDNOT 4340.04  ; INSULATION  TEST START
OUT W38.05  ; INSULATION TEST STOP
; rung 88: CONDITION PL
LD=(300) E2208 #1  ; INSULATION TEST JUDGMENT RESULT (1:OK,2:NG)
OUT H331.04  ; INSULATION OK
; rung 89
LD=(300) E2208 #2  ; INSULATION TEST JUDGMENT RESULT (1:OK,2:NG)
OUT H331.05  ; INSULATION NG

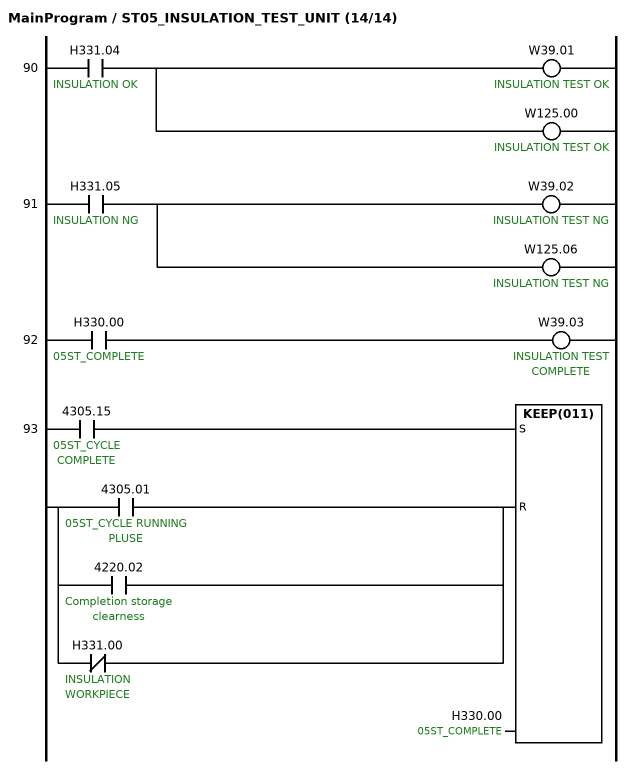
; rung 90
LD H331.04  ; INSULATION OK
OUT W39.01  ; INSULATION TEST OK
OUT W125.00  ; INSULATION TEST OK
; rung 91
LD H331.05  ; INSULATION NG
OUT W39.02  ; INSULATION TEST NG
OUT W125.06  ; INSULATION TEST NG
; rung 92
LD H330.00  ; 05ST_COMPLETE
OUT W39.03  ; INSULATION TEST COMPLETE
; rung 93
LD 4305.15  ; 05ST_CYCLE COMPLETE
LD 4305.01  ; 05ST_CYCLE RUNNING PLUSE
OR 4220.02  ; Completion storage clearness
ORNOT H331.00  ; INSULATION WORKPIECE
KEEP(011) H330.00  ; 05ST_COMPLETE

### Section ST06_SWING_MEASURE_UNIT

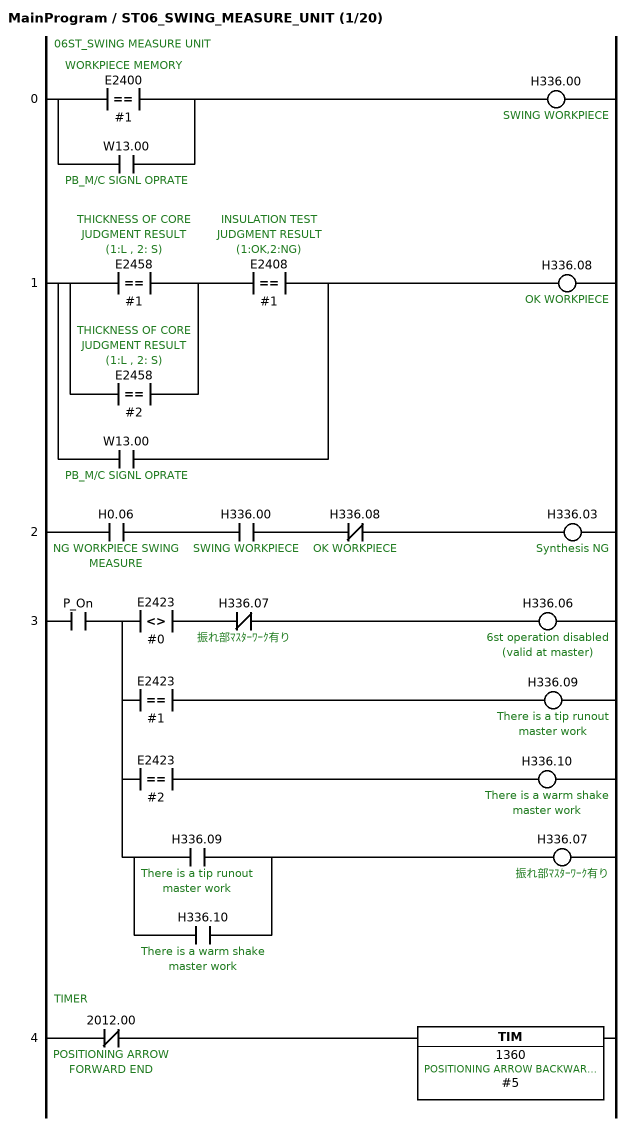
; rung 0: 06ST_SWING MEASURE UNIT
LD=(300) E2400 #1  ; WORKPIECE MEMORY
OR W13.00  ; PB_M/C SIGNL OPRATE
OUT H336.00  ; SWING WORKPIECE
; rung 1
LD=(300) E2458 #1  ; THICKNESS OF CORE JUDGMENT RESULT (1:L , 2: S)
OR=(300) E2458 #2  ; THICKNESS OF CORE JUDGMENT RESULT (1:L , 2: S)
AND=(300) E2408 #1  ; INSULATION TEST JUDGMENT RESULT (1:OK,2:NG)
OR W13.00  ; PB_M/C SIGNL OPRATE
OUT H336.08  ; OK WORKPIECE
; rung 2
LD H0.06  ; NG WORKPIECE SWING MEASURE
AND H336.00  ; SWING WORKPIECE
ANDNOT H336.08  ; OK WORKPIECE
OUT H336.03  ; Synthesis NG
; rung 3
LD P_On
OUT TR0
AND<>(305) E2423 #0
ANDNOT H336.07  ; 振れ部ﾏｽﾀｰﾜｰｸ有り
OUT H336.06  ; 6st operation disabled (valid at master)
LD TR0
AND=(300) E2423 #1
OUT H336.09  ; There is a tip runout master work
LD TR0
AND=(300) E2423 #2
OUT H336.10  ; There is a warm shake master work
LD TR0
LD H336.09  ; There is a tip runout master work
OR H336.10  ; There is a warm shake master work
ANDLD
OUT H336.07  ; 振れ部ﾏｽﾀｰﾜｰｸ有り
; rung 4: TIMER
LDNOT 2012.00  ; POSITIONING ARROW FORWARD END
TIM 1360 #5  ; POSITIONING ARROW BACKWARD END

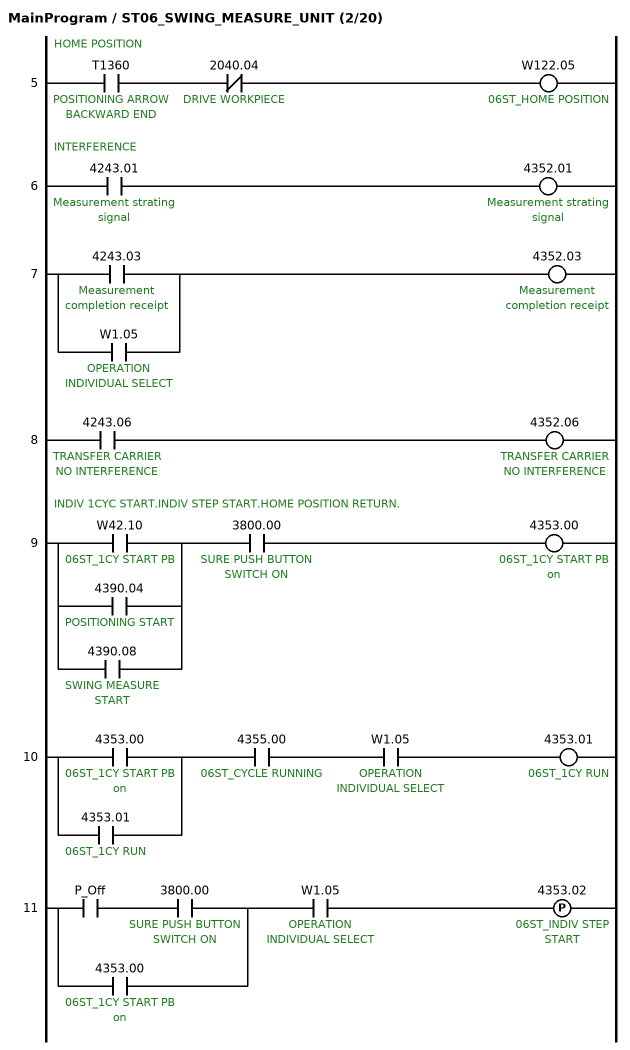
; rung 5: HOME POSITION
LD T1360  ; POSITIONING ARROW BACKWARD END
ANDNOT 2040.04  ; DRIVE WORKPIECE
OUT W122.05  ; 06ST_HOME POSITION
; rung 6: INTERFERENCE
LD 4243.01  ; Measurement strating signal
OUT 4352.01  ; Measurement strating signal
; rung 7
LD 4243.03  ; Measurement completion receipt
OR W1.05  ; OPERATION INDIVIDUAL SELECT
OUT 4352.03  ; Measurement completion receipt
; rung 8
LD 4243.06  ; TRANSFER CARRIER NO INTERFERENCE
OUT 4352.06  ; TRANSFER CARRIER NO INTERFERENCE
; rung 9: INDIV 1CYC START.INDIV STEP START.HOME POSITION RETURN.
LD W42.10  ; 06ST_1CY START PB
OR 4390.04  ; POSITIONING START
OR 4390.08  ; SWING MEASURE START
AND 3800.00  ; SURE PUSH BUTTON SWITCH ON
OUT 4353.00  ; 06ST_1CY START PB on
; rung 10
LD 4353.00  ; 06ST_1CY START PB on
OR 4353.01  ; 06ST_1CY RUN
AND 4355.00  ; 06ST_CYCLE RUNNING
AND W1.05  ; OPERATION INDIVIDUAL SELECT
OUT 4353.01  ; 06ST_1CY RUN
; rung 11
LD P_Off
AND 3800.00  ; SURE PUSH BUTTON SWITCH ON
OR 4353.00  ; 06ST_1CY START PB on
AND W1.05  ; OPERATION INDIVIDUAL SELECT
DIFU(013) 4353.02  ; 06ST_INDIV STEP START

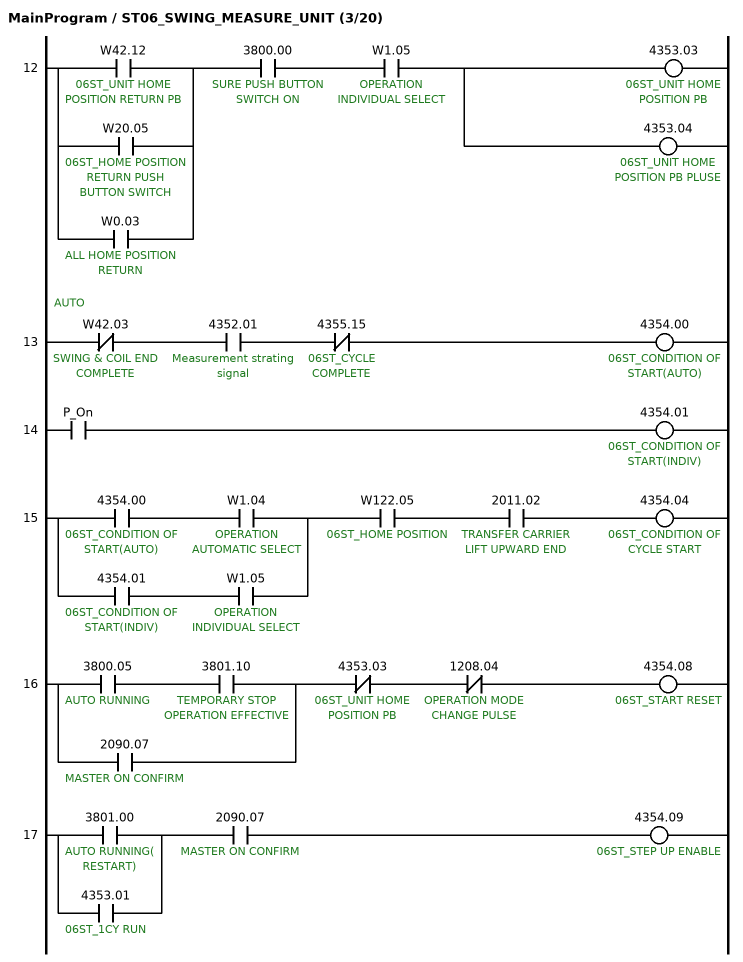
; rung 12
LD W42.12  ; 06ST_UNIT HOME POSITION RETURN PB
OR W20.05  ; 06ST_HOME POSITION RETURN PUSH BUTTON SWITCH
OR W0.03  ; ALL HOME POSITION RETURN
AND 3800.00  ; SURE PUSH BUTTON SWITCH ON
AND W1.05  ; OPERATION INDIVIDUAL SELECT
OUT 4353.03  ; 06ST_UNIT HOME POSITION PB
OUT 4353.04  ; 06ST_UNIT HOME POSITION PB PLUSE
; rung 13: AUTO
LDNOT W42.03  ; SWING & COIL END COMPLETE
AND 4352.01  ; Measurement strating signal
ANDNOT 4355.15  ; 06ST_CYCLE COMPLETE
OUT 4354.00  ; 06ST_CONDITION OF START(AUTO)
; rung 14
LD P_On
OUT 4354.01  ; 06ST_CONDITION OF START(INDIV)
; rung 15
LD 4354.00  ; 06ST_CONDITION OF START(AUTO)
AND W1.04  ; OPERATION AUTOMATIC SELECT
LD 4354.01  ; 06ST_CONDITION OF START(INDIV)
AND W1.05  ; OPERATION INDIVIDUAL SELECT
ORLD
AND W122.05  ; 06ST_HOME POSITION
AND 2011.02  ; TRANSFER CARRIER LIFT UPWARD END
OUT 4354.04  ; 06ST_CONDITION OF CYCLE START
; rung 16
LD 3800.05  ; AUTO RUNNING
AND 3801.10  ; TEMPORARY STOP OPERATION EFFECTIVE
OR 2090.07  ; MASTER ON CONFIRM
ANDNOT 4353.03  ; 06ST_UNIT HOME POSITION PB
ANDNOT 1208.04  ; OPERATION MODE CHANGE PULSE
OUT 4354.08  ; 06ST_START RESET
; rung 17
LD 3801.00  ; AUTO RUNNING(RESTART)
OR 4353.01  ; 06ST_1CY RUN
AND 2090.07  ; MASTER ON CONFIRM
OUT 4354.09  ; 06ST_STEP UP ENABLE

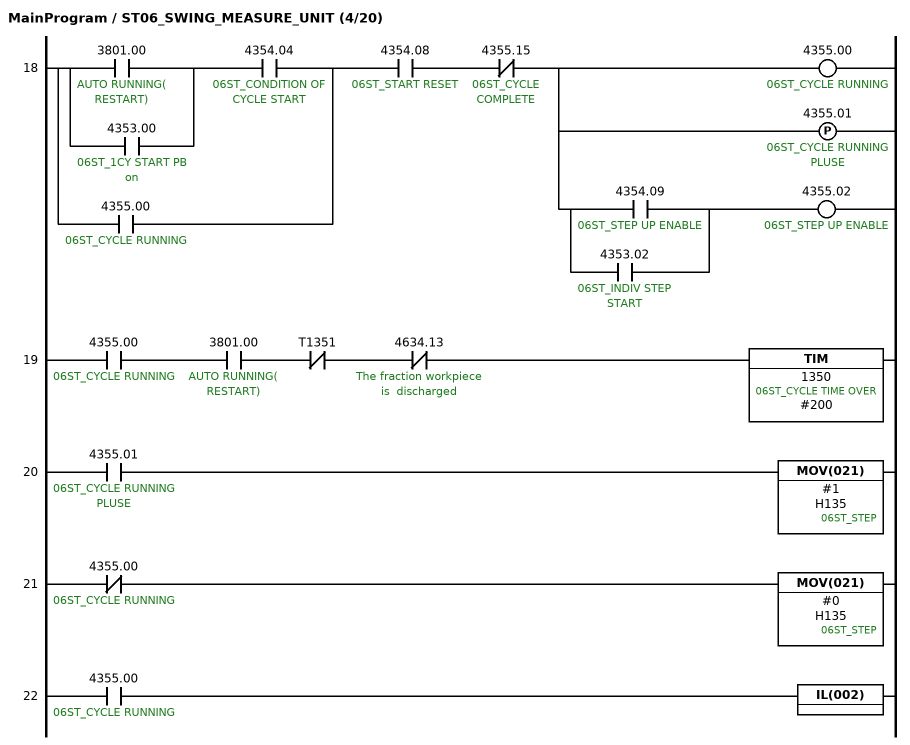
; rung 18
LD 3801.00  ; AUTO RUNNING(RESTART)
OR 4353.00  ; 06ST_1CY START PB on
AND 4354.04  ; 06ST_CONDITION OF CYCLE START
OR 4355.00  ; 06ST_CYCLE RUNNING
AND 4354.08  ; 06ST_START RESET
ANDNOT 4355.15  ; 06ST_CYCLE COMPLETE
OUT 4355.00  ; 06ST_CYCLE RUNNING
DIFU(013) 4355.01  ; 06ST_CYCLE RUNNING PLUSE
LD 4354.09  ; 06ST_STEP UP ENABLE
OR 4353.02  ; 06ST_INDIV STEP START
ANDLD
OUT 4355.02  ; 06ST_STEP UP ENABLE
; rung 19
LD 4355.00  ; 06ST_CYCLE RUNNING
AND 3801.00  ; AUTO RUNNING(RESTART)
ANDNOT T1351
ANDNOT 4634.13  ; The fraction workpiece is  discharged
TIM 1350 #200  ; 06ST_CYCLE TIME OVER
; rung 20
LD 4355.01  ; 06ST_CYCLE RUNNING PLUSE
MOV(021) #1 H135  ; 06ST_STEP
; rung 21
LDNOT 4355.00  ; 06ST_CYCLE RUNNING
MOV(021) #0 H135  ; 06ST_STEP
; rung 22
LD 4355.00  ; 06ST_CYCLE RUNNING
IL(002)

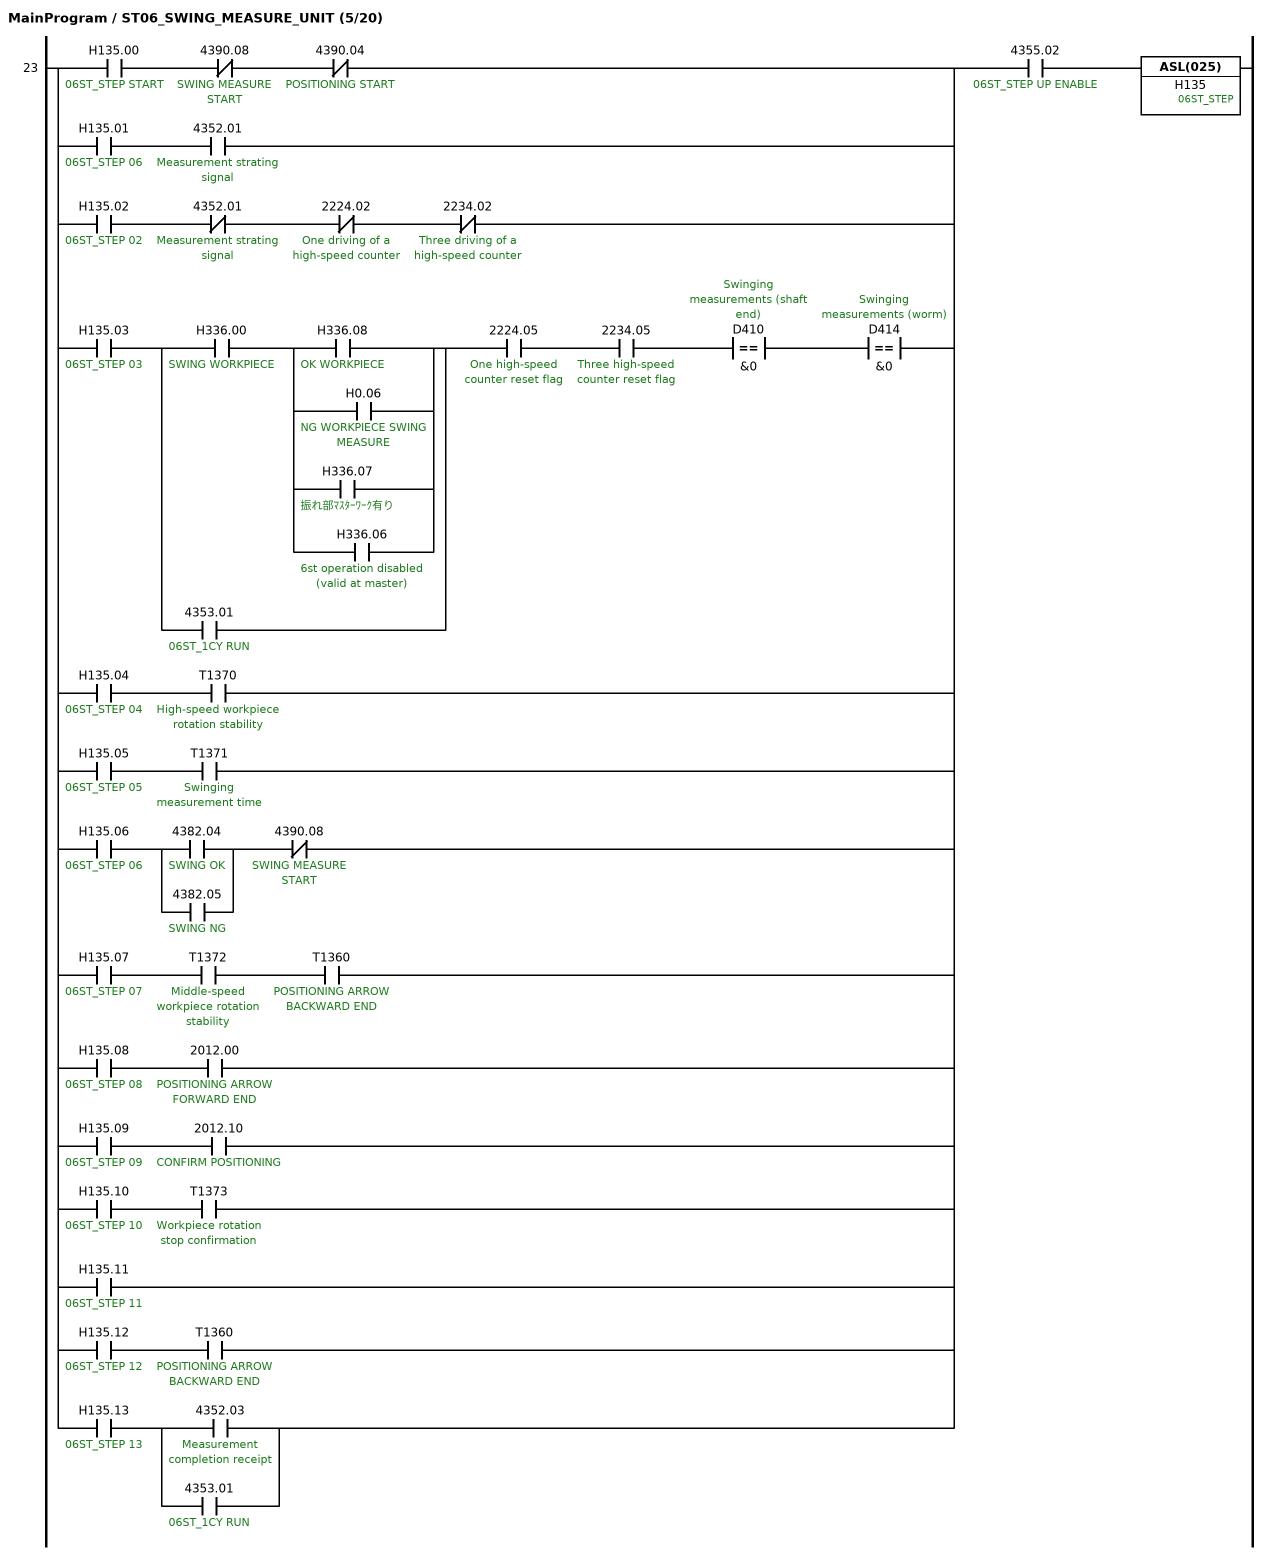
; rung 23
LD H135.00  ; 06ST_STEP START
ANDNOT 4390.08  ; SWING MEASURE START
ANDNOT 4390.04  ; POSITIONING START
LD H135.01  ; 06ST_STEP 06
AND 4352.01  ; Measurement strating signal
ORLD
LD H135.02  ; 06ST_STEP 02
ANDNOT 4352.01  ; Measurement strating signal
ANDNOT 2224.02  ; One driving of a high-speed counter
ANDNOT 2234.02  ; Three driving of a high-speed counter
ORLD
LD H135.03  ; 06ST_STEP 03
LD H336.00  ; SWING WORKPIECE
LD H336.08  ; OK WORKPIECE
OR H0.06  ; NG WORKPIECE SWING MEASURE
OR H336.07  ; 振れ部ﾏｽﾀｰﾜｰｸ有り
OR H336.06  ; 6st operation disabled (valid at master)
ANDLD
OR 4353.01  ; 06ST_1CY RUN
ANDLD
AND 2224.05  ; One high-speed counter reset flag
AND 2234.05  ; Three high-speed counter reset flag
AND=(300) D410 &0  ; Swinging measurements (shaft end)
AND=(300) D414 &0  ; Swinging measurements (worm)
ORLD
LD H135.04  ; 06ST_STEP 04
AND T1370  ; High-speed workpiece rotation stability
ORLD
LD H135.05  ; 06ST_STEP 05
AND T1371  ; Swinging measurement time
ORLD
LD H135.06  ; 06ST_STEP 06
LD 4382.04  ; SWING OK
OR 4382.05  ; SWING NG
ANDLD
ANDNOT 4390.08  ; SWING MEASURE START
ORLD
LD H135.07  ; 06ST_STEP 07
AND T1372  ; Middle-speed workpiece rotation stability
AND T1360  ; POSITIONING ARROW BACKWARD END
ORLD
LD H135.08  ; 06ST_STEP 08
AND 2012.00  ; POSITIONING ARROW FORWARD END
ORLD
LD H135.09  ; 06ST_STEP 09
AND 2012.10  ; CONFIRM POSITIONING
ORLD
LD H135.10  ; 06ST_STEP 10
AND T1373  ; Workpiece rotation stop confirmation
ORLD
OR H135.11  ; 06ST_STEP 11
LD H135.12  ; 06ST_STEP 12
AND T1360  ; POSITIONING ARROW BACKWARD END
ORLD
LD H135.13  ; 06ST_STEP 13
LD 4352.03  ; Measurement completion receipt
OR 4353.01  ; 06ST_1CY RUN
ANDLD
ORLD
AND 4355.02  ; 06ST_STEP UP ENABLE
ASL(025) H135  ; 06ST_STEP

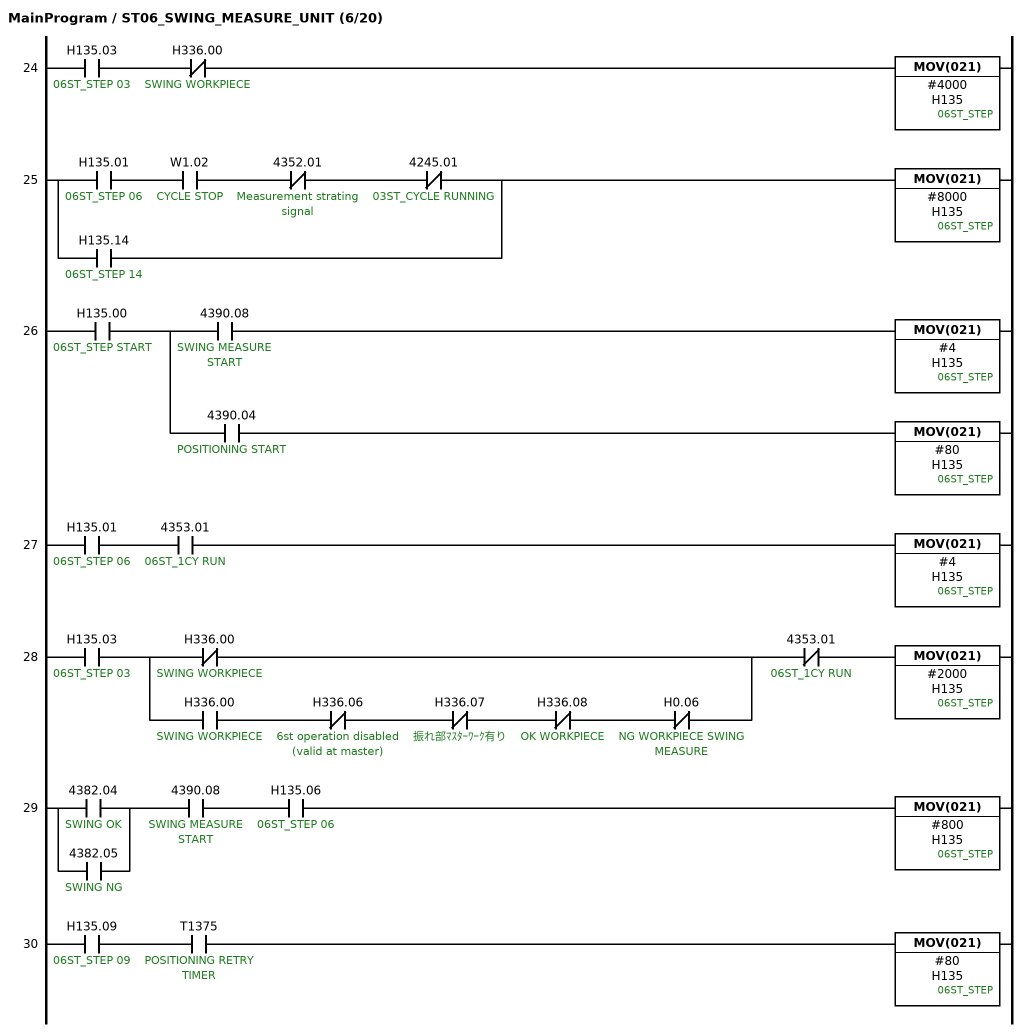
; rung 24
LD H135.03  ; 06ST_STEP 03
ANDNOT H336.00  ; SWING WORKPIECE
MOV(021) #4000 H135  ; 06ST_STEP
; rung 25
LD H135.01  ; 06ST_STEP 06
AND W1.02  ; CYCLE STOP
ANDNOT 4352.01  ; Measurement strating signal
ANDNOT 4245.01  ; 03ST_CYCLE RUNNING
OR H135.14  ; 06ST_STEP 14
MOV(021) #8000 H135  ; 06ST_STEP
; rung 26
LD H135.00  ; 06ST_STEP START
OUT TR0
AND 4390.08  ; SWING MEASURE START
MOV(021) #4 H135  ; 06ST_STEP
LD TR0
AND 4390.04  ; POSITIONING START
MOV(021) #80 H135  ; 06ST_STEP
; rung 27
LD H135.01  ; 06ST_STEP 06
AND 4353.01  ; 06ST_1CY RUN
MOV(021) #4 H135  ; 06ST_STEP
; rung 28
LD H135.03  ; 06ST_STEP 03
LDNOT H336.00  ; SWING WORKPIECE
LD H336.00  ; SWING WORKPIECE
ANDNOT H336.06  ; 6st operation disabled (valid at master)
ANDNOT H336.07  ; 振れ部ﾏｽﾀｰﾜｰｸ有り
ANDNOT H336.08  ; OK WORKPIECE
ANDNOT H0.06  ; NG WORKPIECE SWING MEASURE
ORLD
ANDLD
ANDNOT 4353.01  ; 06ST_1CY RUN
MOV(021) #2000 H135  ; 06ST_STEP
; rung 29
LD 4382.04  ; SWING OK
OR 4382.05  ; SWING NG
AND 4390.08  ; SWING MEASURE START
AND H135.06  ; 06ST_STEP 06
MOV(021) #800 H135  ; 06ST_STEP
; rung 30
LD H135.09  ; 06ST_STEP 09
AND T1375  ; POSITIONING RETRY TIMER
MOV(021) #80 H135  ; 06ST_STEP

